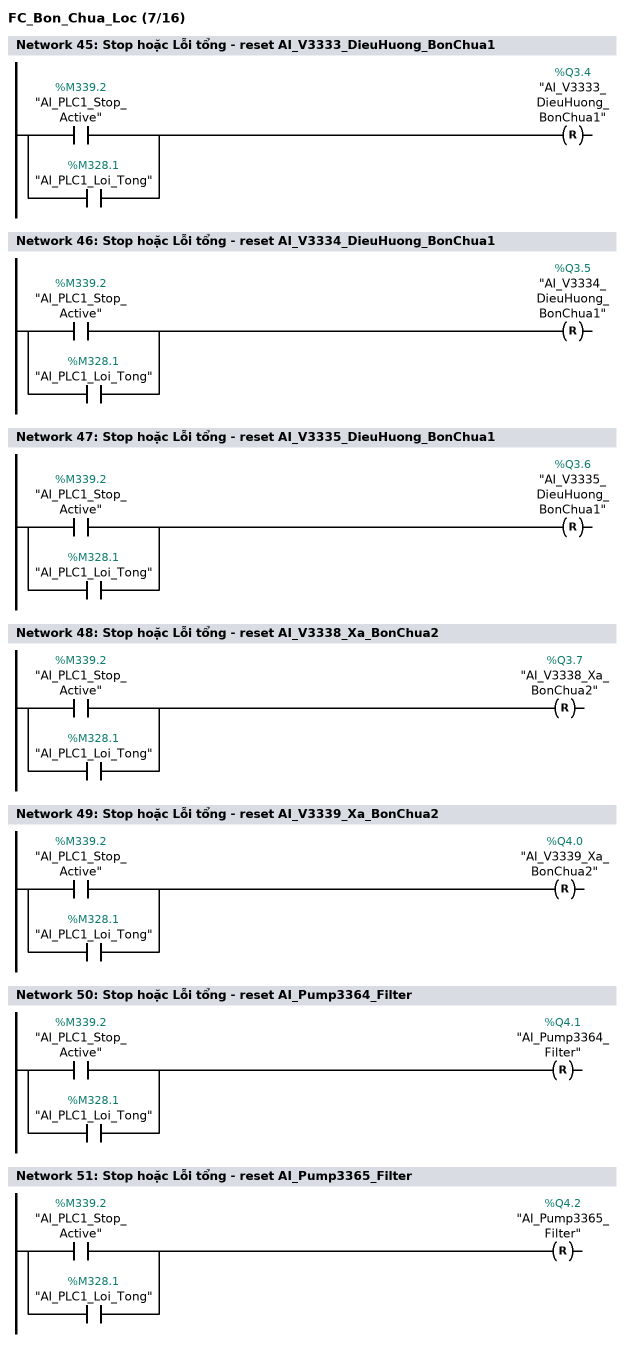
   RUNG wire#powerrail
      Contact( "AI_PLC1_Stop_Active" )
      wire#w1
      R_Coil( "AI_V3333_DieuHuong_BonChua1" )
   END_RUNG
   RUNG wire#powerrail
      Contact( "AI_PLC1_Loi_Tong" )
   END_RUNG wire#w1
   // the same network as SCL:
   IF "AI_PLC1_Stop_Active" OR "AI_PLC1_Loi_Tong" THEN "AI_V3333_DieuHuong_BonChua1" := FALSE; END_IF;
END_REGION

REGION Network 46: Stop hoặc Lỗi tổng - reset AI_V3334_DieuHuong_BonChua1
   RUNG wire#powerrail
      Contact( "AI_PLC1_Stop_Active" )
      wire#w1
      R_Coil( "AI_V3334_DieuHuong_BonChua1" )
   END_RUNG
   RUNG wire#powerrail
      Contact( "AI_PLC1_Loi_Tong" )
   END_RUNG wire#w1
   // the same network as SCL:
   IF "AI_PLC1_Stop_Active" OR "AI_PLC1_Loi_Tong" THEN "AI_V3334_DieuHuong_BonChua1" := FALSE; END_IF;
END_REGION

REGION Network 47: Stop hoặc Lỗi tổng - reset AI_V3335_DieuHuong_BonChua1
   RUNG wire#powerrail
      Contact( "AI_PLC1_Stop_Active" )
      wire#w1
      R_Coil( "AI_V3335_DieuHuong_BonChua1" )
   END_RUNG
   RUNG wire#powerrail
      Contact( "AI_PLC1_Loi_Tong" )
   END_RUNG wire#w1
   // the same network as SCL:
   IF "AI_PLC1_Stop_Active" OR "AI_PLC1_Loi_Tong" THEN "AI_V3335_DieuHuong_BonChua1" := FALSE; END_IF;
END_REGION

REGION Network 48: Stop hoặc Lỗi tổng - reset AI_V3338_Xa_BonChua2
   RUNG wire#powerrail
      Contact( "AI_PLC1_Stop_Active" )
      wire#w1
      R_Coil( "AI_V3338_Xa_BonChua2" )
   END_RUNG
   RUNG wire#powerrail
      Contact( "AI_PLC1_Loi_Tong" )
   END_RUNG wire#w1
   // the same network as SCL:
   IF "AI_PLC1_Stop_Active" OR "AI_PLC1_Loi_Tong" THEN "AI_V3338_Xa_BonChua2" := FALSE; END_IF;
END_REGION

REGION Network 49: Stop hoặc Lỗi tổng - reset AI_V3339_Xa_BonChua2
   RUNG wire#powerrail
      Contact( "AI_PLC1_Stop_Active" )
      wire#w1
      R_Coil( "AI_V3339_Xa_BonChua2" )
   END_RUNG
   RUNG wire#powerrail
      Contact( "AI_PLC1_Loi_Tong" )
   END_RUNG wire#w1
   // the same network as SCL:
   IF "AI_PLC1_Stop_Active" OR "AI_PLC1_Loi_Tong" THEN "AI_V3339_Xa_BonChua2" := FALSE; END_IF;
END_REGION

REGION Network 50: Stop hoặc Lỗi tổng - reset AI_Pump3364_Filter
   RUNG wire#powerrail
      Contact( "AI_PLC1_Stop_Active" )
      wire#w1
      R_Coil( "AI_Pump3364_Filter" )
   END_RUNG
   RUNG wire#powerrail
      Contact( "AI_PLC1_Loi_Tong" )
   END_RUNG wire#w1
   // the same network as SCL:
   IF "AI_PLC1_Stop_Active" OR "AI_PLC1_Loi_Tong" THEN "AI_Pump3364_Filter" := FALSE; END_IF;
END_REGION

REGION Network 51: Stop hoặc Lỗi tổng - reset AI_Pump3365_Filter
   RUNG wire#powerrail
      Contact( "AI_PLC1_Stop_Active" )
      wire#w1
      R_Coil( "AI_Pump3365_Filter" )
   END_RUNG
   RUNG wire#powerrail
      Contact( "AI_PLC1_Loi_Tong" )
   END_RUNG wire#w1
   // the same network as SCL:
   IF "AI_PLC1_Stop_Active" OR "AI_PLC1_Loi_Tong" THEN "AI_Pump3365_Filter" := FALSE; END_IF;
END_REGION

REGION Network 52: Stop hoặc Lỗi tổng - reset AI_V3340_Duong_Filter
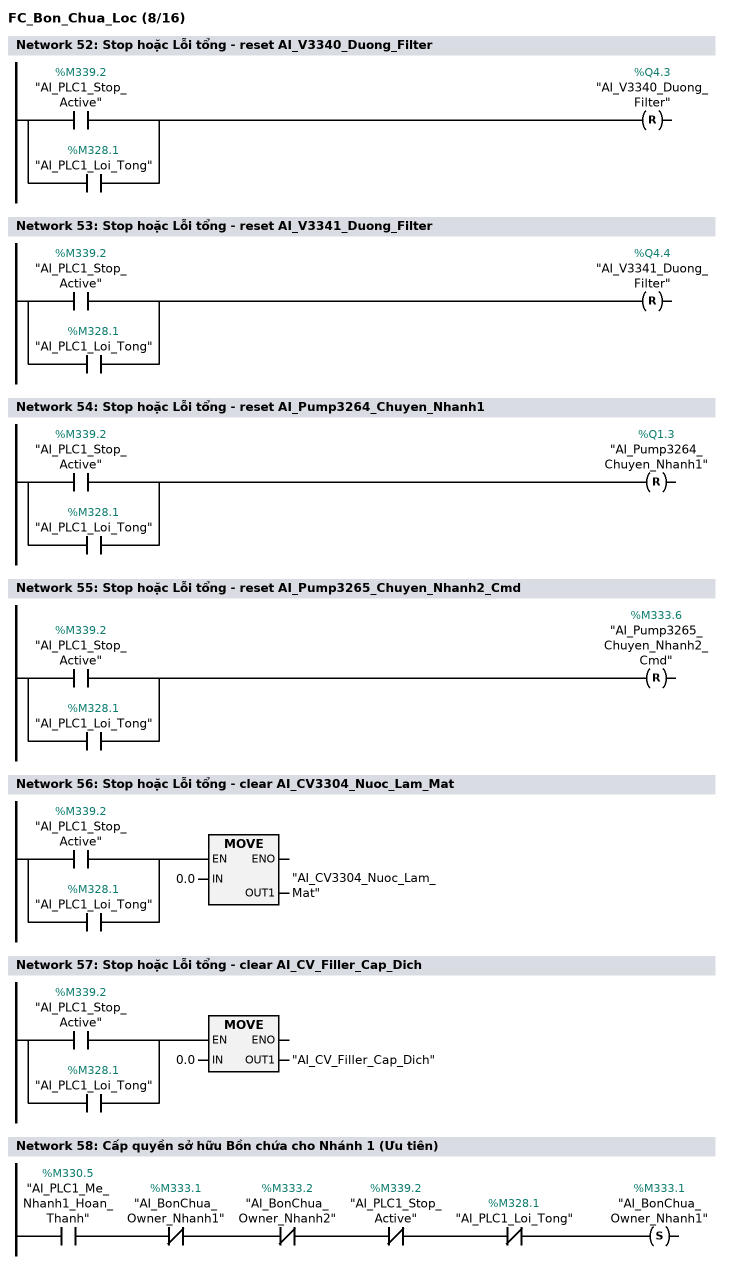
   RUNG wire#powerrail
      Contact( "AI_PLC1_Stop_Active" )
      wire#w1
      R_Coil( "AI_V3340_Duong_Filter" )
   END_RUNG
   RUNG wire#powerrail
      Contact( "AI_PLC1_Loi_Tong" )
   END_RUNG wire#w1
   // the same network as SCL:
   IF "AI_PLC1_Stop_Active" OR "AI_PLC1_Loi_Tong" THEN "AI_V3340_Duong_Filter" := FALSE; END_IF;
END_REGION

REGION Network 53: Stop hoặc Lỗi tổng - reset AI_V3341_Duong_Filter
   RUNG wire#powerrail
      Contact( "AI_PLC1_Stop_Active" )
      wire#w1
      R_Coil( "AI_V3341_Duong_Filter" )
   END_RUNG
   RUNG wire#powerrail
      Contact( "AI_PLC1_Loi_Tong" )
   END_RUNG wire#w1
   // the same network as SCL:
   IF "AI_PLC1_Stop_Active" OR "AI_PLC1_Loi_Tong" THEN "AI_V3341_Duong_Filter" := FALSE; END_IF;
END_REGION

REGION Network 54: Stop hoặc Lỗi tổng - reset AI_Pump3264_Chuyen_Nhanh1
   RUNG wire#powerrail
      Contact( "AI_PLC1_Stop_Active" )
      wire#w1
      R_Coil( "AI_Pump3264_Chuyen_Nhanh1" )
   END_RUNG
   RUNG wire#powerrail
      Contact( "AI_PLC1_Loi_Tong" )
   END_RUNG wire#w1
   // the same network as SCL:
   IF "AI_PLC1_Stop_Active" OR "AI_PLC1_Loi_Tong" THEN "AI_Pump3264_Chuyen_Nhanh1" := FALSE; END_IF;
END_REGION

REGION Network 55: Stop hoặc Lỗi tổng - reset AI_Pump3265_Chuyen_Nhanh2_Cmd
   RUNG wire#powerrail
      Contact( "AI_PLC1_Stop_Active" )
      wire#w1
      R_Coil( "AI_Pump3265_Chuyen_Nhanh2_Cmd" )
   END_RUNG
   RUNG wire#powerrail
      Contact( "AI_PLC1_Loi_Tong" )
   END_RUNG wire#w1
   // the same network as SCL:
   IF "AI_PLC1_Stop_Active" OR "AI_PLC1_Loi_Tong" THEN "AI_Pump3265_Chuyen_Nhanh2_Cmd" := FALSE; END_IF;
END_REGION

REGION Network 56: Stop hoặc Lỗi tổng - clear AI_CV3304_Nuoc_Lam_Mat
   RUNG wire#powerrail
      Contact( "AI_PLC1_Stop_Active" )
      wire#w1
      { S7_GenerateENO := "TRUE" } Move(in := 0.0, out1 => "AI_CV3304_Nuoc_Lam_Mat")
   END_RUNG
   RUNG wire#powerrail
      Contact( "AI_PLC1_Loi_Tong" )
   END_RUNG wire#w1
   // the same network as SCL:
   IF "AI_PLC1_Stop_Active" OR "AI_PLC1_Loi_Tong" THEN "AI_CV3304_Nuoc_Lam_Mat" := 0.0; END_IF;
END_REGION

REGION Network 57: Stop hoặc Lỗi tổng - clear AI_CV_Filler_Cap_Dich
   RUNG wire#powerrail
      Contact( "AI_PLC1_Stop_Active" )
      wire#w1
      { S7_GenerateENO := "TRUE" } Move(in := 0.0, out1 => "AI_CV_Filler_Cap_Dich")
   END_RUNG
   RUNG wire#powerrail
      Contact( "AI_PLC1_Loi_Tong" )
   END_RUNG wire#w1
   // the same network as SCL:
   IF "AI_PLC1_Stop_Active" OR "AI_PLC1_Loi_Tong" THEN "AI_CV_Filler_Cap_Dich" := 0.0; END_IF;
END_REGION

REGION Network 58: Cấp quyền sở hữu Bồn chứa cho Nhánh 1 (Ưu tiên)
   RUNG wire#powerrail
      Contact( "AI_PLC1_Me_Nhanh1_Hoan_Thanh" )
      I_Contact( "AI_BonChua_Owner_Nhanh1" )
      I_Contact( "AI_BonChua_Owner_Nhanh2" )
      I_Contact( "AI_PLC1_Stop_Active" )
      I_Contact( "AI_PLC1_Loi_Tong" )
      S_Coil( "AI_BonChua_Owner_Nhanh1" )
   END_RUNG
   // the same network as SCL:
   IF "AI_PLC1_Me_Nhanh1_Hoan_Thanh" AND NOT "AI_BonChua_Owner_Nhanh1" AND NOT "AI_BonChua_Owner_Nhanh2" AND NOT "AI_PLC1_Stop_Active" AND NOT "AI_PLC1_Loi_Tong" THEN
       "AI_BonChua_Owner_Nhanh1" := TRUE;
   END_IF;
END_REGION

REGION Network 59: Cấp quyền sở hữu Bồn chứa cho Nhánh 2
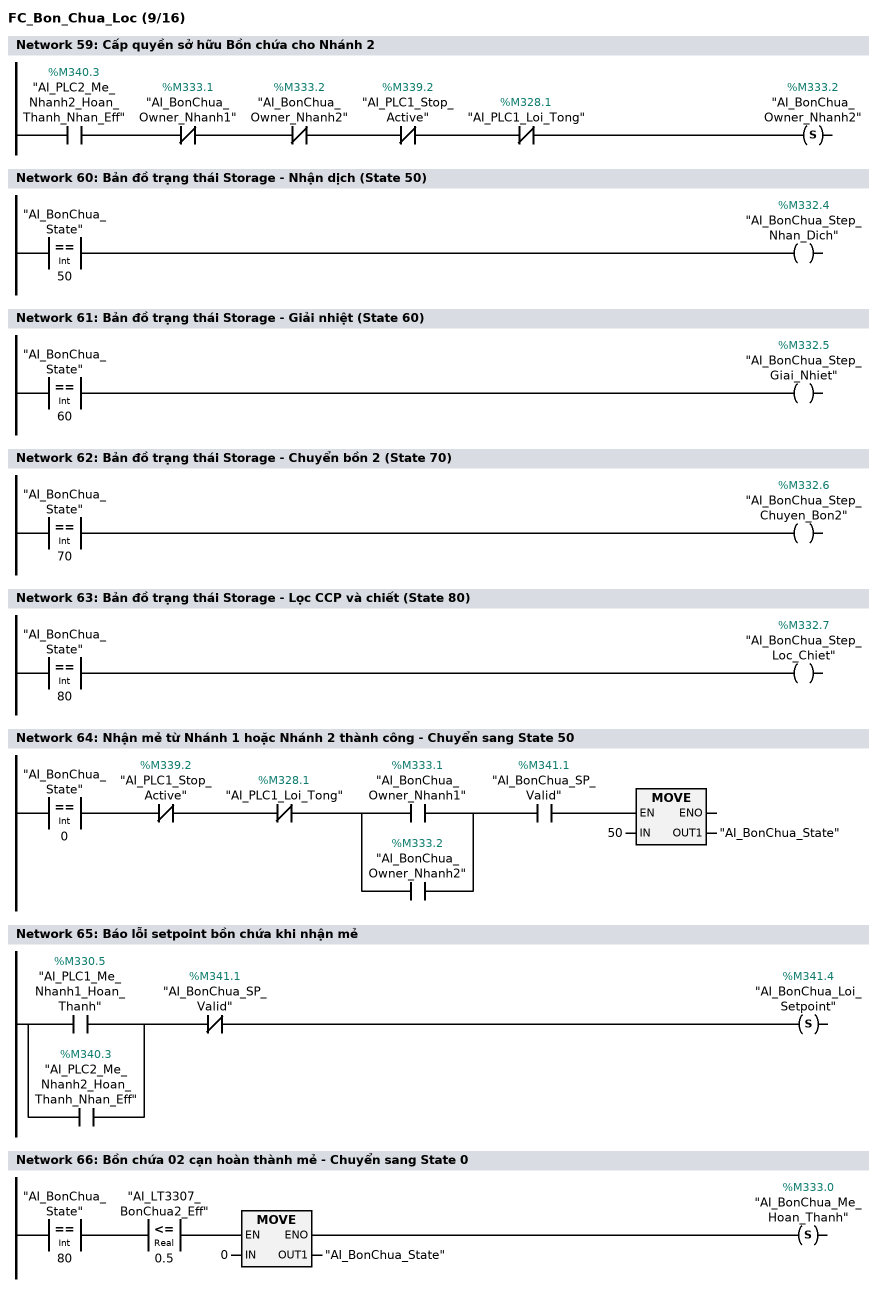
   RUNG wire#powerrail
      Contact( "AI_PLC2_Me_Nhanh2_Hoan_Thanh_Nhan_Eff" )
      I_Contact( "AI_BonChua_Owner_Nhanh1" )
      I_Contact( "AI_BonChua_Owner_Nhanh2" )
      I_Contact( "AI_PLC1_Stop_Active" )
      I_Contact( "AI_PLC1_Loi_Tong" )
      S_Coil( "AI_BonChua_Owner_Nhanh2" )
   END_RUNG
   // the same network as SCL:
   IF "AI_PLC2_Me_Nhanh2_Hoan_Thanh_Nhan_Eff" AND NOT "AI_BonChua_Owner_Nhanh1" AND NOT "AI_BonChua_Owner_Nhanh2" AND NOT "AI_PLC1_Stop_Active" AND NOT "AI_PLC1_Loi_Tong" THEN
       "AI_BonChua_Owner_Nhanh2" := TRUE;
   END_IF;
END_REGION

REGION Network 60: Bản đồ trạng thái Storage - Nhận dịch (State 50)
   RUNG wire#powerrail
      { S7_Templates := "SrcType := Int" } EQ_Contact(in1 := "AI_BonChua_State", in2 := 50)
      Coil( "AI_BonChua_Step_Nhan_Dich" )
   END_RUNG
   // the same network as SCL:
   "AI_BonChua_Step_Nhan_Dich" := "AI_BonChua_State" = 50;
END_REGION

REGION Network 61: Bản đồ trạng thái Storage - Giải nhiệt (State 60)
   RUNG wire#powerrail
      { S7_Templates := "SrcType := Int" } EQ_Contact(in1 := "AI_BonChua_State", in2 := 60)
      Coil( "AI_BonChua_Step_Giai_Nhiet" )
   END_RUNG
   // the same network as SCL:
   "AI_BonChua_Step_Giai_Nhiet" := "AI_BonChua_State" = 60;
END_REGION

REGION Network 62: Bản đồ trạng thái Storage - Chuyển bồn 2 (State 70)
   RUNG wire#powerrail
      { S7_Templates := "SrcType := Int" } EQ_Contact(in1 := "AI_BonChua_State", in2 := 70)
      Coil( "AI_BonChua_Step_Chuyen_Bon2" )
   END_RUNG
   // the same network as SCL:
   "AI_BonChua_Step_Chuyen_Bon2" := "AI_BonChua_State" = 70;
END_REGION

REGION Network 63: Bản đồ trạng thái Storage - Lọc CCP và chiết (State 80)
   RUNG wire#powerrail
      { S7_Templates := "SrcType := Int" } EQ_Contact(in1 := "AI_BonChua_State", in2 := 80)
      Coil( "AI_BonChua_Step_Loc_Chiet" )
   END_RUNG
   // the same network as SCL:
   "AI_BonChua_Step_Loc_Chiet" := "AI_BonChua_State" = 80;
END_REGION

REGION Network 64: Nhận mẻ từ Nhánh 1 hoặc Nhánh 2 thành công - Chuyển sang State 50
   RUNG wire#powerrail
      { S7_Templates := "SrcType := Int" } EQ_Contact(in1 := "AI_BonChua_State", in2 := 0)
      I_Contact( "AI_PLC1_Stop_Active" )
      I_Contact( "AI_PLC1_Loi_Tong" )
      wire#w1
      Contact( "AI_BonChua_Owner_Nhanh1" )
      wire#w2
      Contact( "AI_BonChua_SP_Valid" )
      { S7_GenerateENO := "TRUE" } Move(in := 50, out1 => "AI_BonChua_State")
   END_RUNG
   RUNG wire#w1
      Contact( "AI_BonChua_Owner_Nhanh2" )
   END_RUNG wire#w2
   // the same network as SCL:
   IF ("AI_BonChua_State" = 0) AND NOT "AI_PLC1_Stop_Active" AND NOT "AI_PLC1_Loi_Tong" AND ("AI_BonChua_Owner_Nhanh1" OR "AI_BonChua_Owner_Nhanh2") AND "AI_BonChua_SP_Valid" THEN
       "AI_BonChua_State" := 50;
   END_IF;
END_REGION

REGION Network 65: Báo lỗi setpoint bồn chứa khi nhận mẻ
   RUNG wire#powerrail
      Contact( "AI_PLC1_Me_Nhanh1_Hoan_Thanh" )
      wire#w1
      I_Contact( "AI_BonChua_SP_Valid" )
      S_Coil( "AI_BonChua_Loi_Setpoint" )
   END_RUNG
   RUNG wire#powerrail
      Contact( "AI_PLC2_Me_Nhanh2_Hoan_Thanh_Nhan_Eff" )
   END_RUNG wire#w1
   // the same network as SCL:
   IF ("AI_PLC1_Me_Nhanh1_Hoan_Thanh" OR "AI_PLC2_Me_Nhanh2_Hoan_Thanh_Nhan_Eff") AND NOT "AI_BonChua_SP_Valid" THEN
       "AI_BonChua_Loi_Setpoint" := TRUE;
   END_IF;
END_REGION

REGION Network 66: Bồn chứa 02 cạn hoàn thành mẻ - Chuyển sang State 0
   RUNG wire#powerrail
      { S7_Templates := "SrcType := Int" } EQ_Contact(in1 := "AI_BonChua_State", in2 := 80)
      { S7_Templates := "SrcType := Real" } LE_Contact(in1 := "AI_LT3307_BonChua2_Eff", in2 := 0.5)
      { S7_GenerateENO := "TRUE" } Move(in := 0, out1 => "AI_BonChua_State")
      S_Coil( "AI_BonChua_Me_Hoan_Thanh" )
   END_RUNG
   // the same network as SCL:
   // ENO of a box is taken as its EN; it also drops when the box reports an error
   #_w1 := ("AI_BonChua_State" = 80) AND ("AI_LT3307_BonChua2_Eff" <= 0.5);
   IF #_w1 THEN
       "AI_BonChua_State" := 0;
       "AI_BonChua_Me_Hoan_Thanh" := TRUE;
   END_IF;
END_REGION

REGION Network 67: Chuyển sang Bồn chứa 02 xong - Chuyển sang State 80
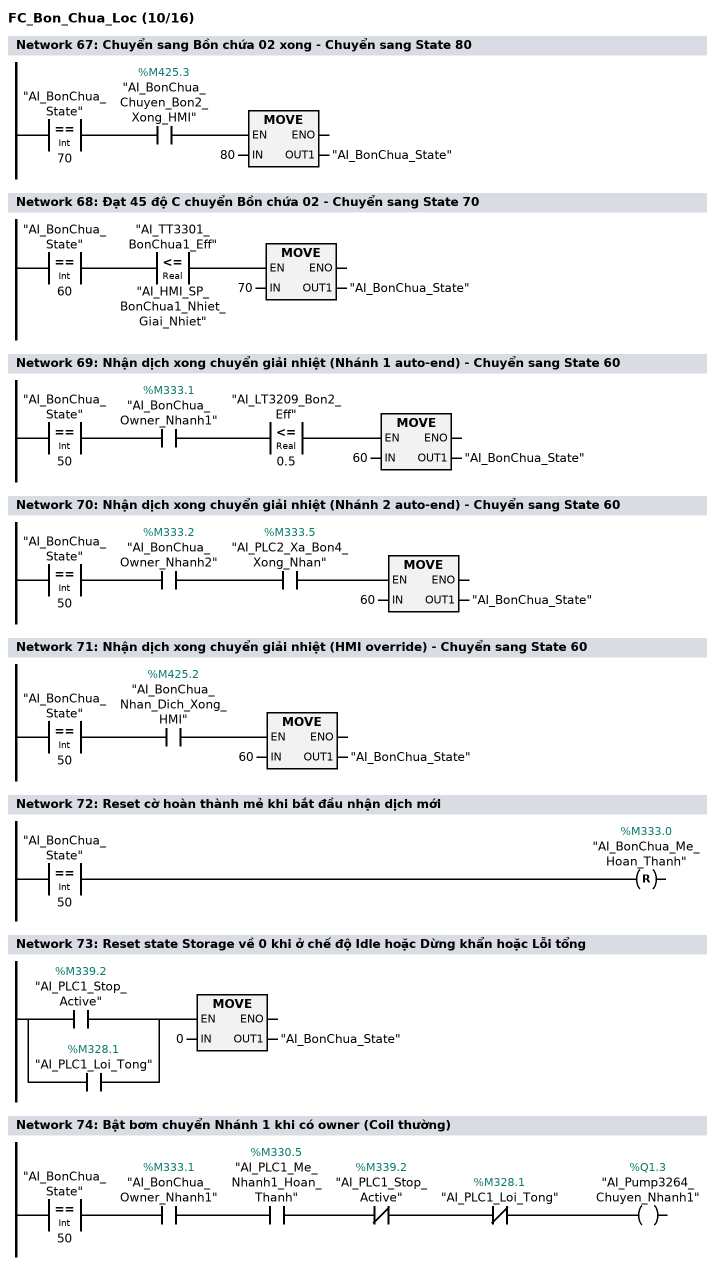
   RUNG wire#powerrail
      { S7_Templates := "SrcType := Int" } EQ_Contact(in1 := "AI_BonChua_State", in2 := 70)
      Contact( "AI_BonChua_Chuyen_Bon2_Xong_HMI" )
      { S7_GenerateENO := "TRUE" } Move(in := 80, out1 => "AI_BonChua_State")
   END_RUNG
   // the same network as SCL:
   IF ("AI_BonChua_State" = 70) AND "AI_BonChua_Chuyen_Bon2_Xong_HMI" THEN "AI_BonChua_State" := 80; END_IF;
END_REGION

REGION Network 68: Đạt 45 độ C chuyển Bồn chứa 02 - Chuyển sang State 70
   RUNG wire#powerrail
      { S7_Templates := "SrcType := Int" } EQ_Contact(in1 := "AI_BonChua_State", in2 := 60)
      { S7_Templates := "SrcType := Real" } LE_Contact(in1 := "AI_TT3301_BonChua1_Eff", in2 := "AI_HMI_SP_BonChua1_Nhiet_Giai_Nhiet")
      { S7_GenerateENO := "TRUE" } Move(in := 70, out1 => "AI_BonChua_State")
   END_RUNG
   // the same network as SCL:
   IF ("AI_BonChua_State" = 60) AND ("AI_TT3301_BonChua1_Eff" <= "AI_HMI_SP_BonChua1_Nhiet_Giai_Nhiet") THEN
       "AI_BonChua_State" := 70;
   END_IF;
END_REGION

REGION Network 69: Nhận dịch xong chuyển giải nhiệt (Nhánh 1 auto-end) - Chuyển sang State 60
   RUNG wire#powerrail
      { S7_Templates := "SrcType := Int" } EQ_Contact(in1 := "AI_BonChua_State", in2 := 50)
      Contact( "AI_BonChua_Owner_Nhanh1" )
      { S7_Templates := "SrcType := Real" } LE_Contact(in1 := "AI_LT3209_Bon2_Eff", in2 := 0.5)
      { S7_GenerateENO := "TRUE" } Move(in := 60, out1 => "AI_BonChua_State")
   END_RUNG
   // the same network as SCL:
   IF ("AI_BonChua_State" = 50) AND "AI_BonChua_Owner_Nhanh1" AND ("AI_LT3209_Bon2_Eff" <= 0.5) THEN
       "AI_BonChua_State" := 60;
   END_IF;
END_REGION

REGION Network 70: Nhận dịch xong chuyển giải nhiệt (Nhánh 2 auto-end) - Chuyển sang State 60
   RUNG wire#powerrail
      { S7_Templates := "SrcType := Int" } EQ_Contact(in1 := "AI_BonChua_State", in2 := 50)
      Contact( "AI_BonChua_Owner_Nhanh2" )
      Contact( "AI_PLC2_Xa_Bon4_Xong_Nhan" )
      { S7_GenerateENO := "TRUE" } Move(in := 60, out1 => "AI_BonChua_State")
   END_RUNG
   // the same network as SCL:
   IF ("AI_BonChua_State" = 50) AND "AI_BonChua_Owner_Nhanh2" AND "AI_PLC2_Xa_Bon4_Xong_Nhan" THEN
       "AI_BonChua_State" := 60;
   END_IF;
END_REGION

REGION Network 71: Nhận dịch xong chuyển giải nhiệt (HMI override) - Chuyển sang State 60
   RUNG wire#powerrail
      { S7_Templates := "SrcType := Int" } EQ_Contact(in1 := "AI_BonChua_State", in2 := 50)
      Contact( "AI_BonChua_Nhan_Dich_Xong_HMI" )
      { S7_GenerateENO := "TRUE" } Move(in := 60, out1 => "AI_BonChua_State")
   END_RUNG
   // the same network as SCL:
   IF ("AI_BonChua_State" = 50) AND "AI_BonChua_Nhan_Dich_Xong_HMI" THEN "AI_BonChua_State" := 60; END_IF;
END_REGION

REGION Network 72: Reset cờ hoàn thành mẻ khi bắt đầu nhận dịch mới
   RUNG wire#powerrail
      { S7_Templates := "SrcType := Int" } EQ_Contact(in1 := "AI_BonChua_State", in2 := 50)
      R_Coil( "AI_BonChua_Me_Hoan_Thanh" )
   END_RUNG
   // the same network as SCL:
   IF "AI_BonChua_State" = 50 THEN "AI_BonChua_Me_Hoan_Thanh" := FALSE; END_IF;
END_REGION

REGION Network 73: Reset state Storage về 0 khi ở chế độ Idle hoặc Dừng khẩn hoặc Lỗi tổng
   RUNG wire#powerrail
      Contact( "AI_PLC1_Stop_Active" )
      wire#w1
      { S7_GenerateENO := "TRUE" } Move(in := 0, out1 => "AI_BonChua_State")
   END_RUNG
   RUNG wire#powerrail
      Contact( "AI_PLC1_Loi_Tong" )
   END_RUNG wire#w1
   // the same network as SCL:
   IF "AI_PLC1_Stop_Active" OR "AI_PLC1_Loi_Tong" THEN "AI_BonChua_State" := 0; END_IF;
END_REGION

REGION Network 74: Bật bơm chuyển Nhánh 1 khi có owner (Coil thường)
   RUNG wire#powerrail
      { S7_Templates := "SrcType := Int" } EQ_Contact(in1 := "AI_BonChua_State", in2 := 50)
      Contact( "AI_BonChua_Owner_Nhanh1" )
      Contact( "AI_PLC1_Me_Nhanh1_Hoan_Thanh" )
      I_Contact( "AI_PLC1_Stop_Active" )
      I_Contact( "AI_PLC1_Loi_Tong" )
      Coil( "AI_Pump3264_Chuyen_Nhanh1" )
   END_RUNG
   // the same network as SCL:
   "AI_Pump3264_Chuyen_Nhanh1" := ("AI_BonChua_State" = 50) AND "AI_BonChua_Owner_Nhanh1" AND "AI_PLC1_Me_Nhanh1_Hoan_Thanh" AND NOT "AI_PLC1_Stop_Active" AND NOT "AI_PLC1_Loi_Tong";
END_REGION

REGION Network 75: Bật bơm chuyển Nhánh 2 khi có owner (Coil thường)
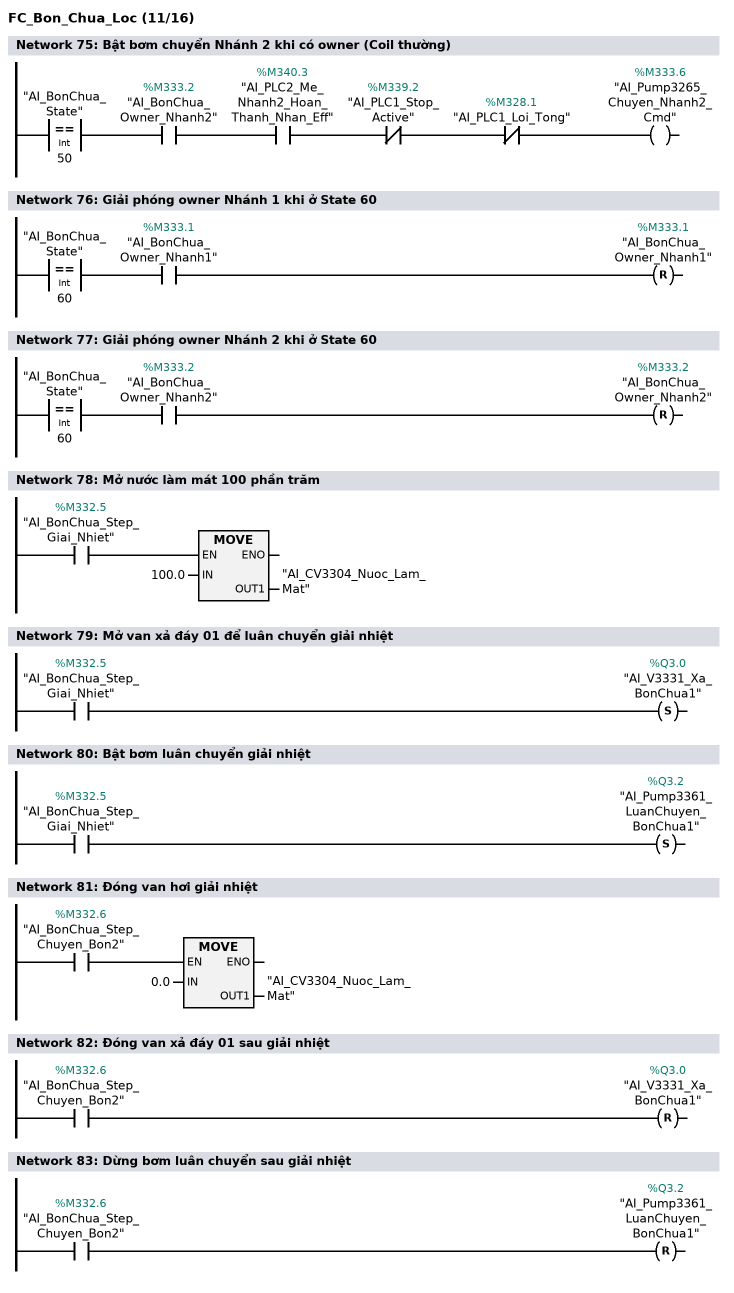
   RUNG wire#powerrail
      { S7_Templates := "SrcType := Int" } EQ_Contact(in1 := "AI_BonChua_State", in2 := 50)
      Contact( "AI_BonChua_Owner_Nhanh2" )
      Contact( "AI_PLC2_Me_Nhanh2_Hoan_Thanh_Nhan_Eff" )
      I_Contact( "AI_PLC1_Stop_Active" )
      I_Contact( "AI_PLC1_Loi_Tong" )
      Coil( "AI_Pump3265_Chuyen_Nhanh2_Cmd" )
   END_RUNG
   // the same network as SCL:
   "AI_Pump3265_Chuyen_Nhanh2_Cmd" := ("AI_BonChua_State" = 50) AND "AI_BonChua_Owner_Nhanh2" AND "AI_PLC2_Me_Nhanh2_Hoan_Thanh_Nhan_Eff" AND NOT "AI_PLC1_Stop_Active" AND NOT "AI_PLC1_Loi_Tong";
END_REGION

REGION Network 76: Giải phóng owner Nhánh 1 khi ở State 60
   RUNG wire#powerrail
      { S7_Templates := "SrcType := Int" } EQ_Contact(in1 := "AI_BonChua_State", in2 := 60)
      Contact( "AI_BonChua_Owner_Nhanh1" )
      R_Coil( "AI_BonChua_Owner_Nhanh1" )
   END_RUNG
   // the same network as SCL:
   IF ("AI_BonChua_State" = 60) AND "AI_BonChua_Owner_Nhanh1" THEN
       "AI_BonChua_Owner_Nhanh1" := FALSE;
   END_IF;
END_REGION

REGION Network 77: Giải phóng owner Nhánh 2 khi ở State 60
   RUNG wire#powerrail
      { S7_Templates := "SrcType := Int" } EQ_Contact(in1 := "AI_BonChua_State", in2 := 60)
      Contact( "AI_BonChua_Owner_Nhanh2" )
      R_Coil( "AI_BonChua_Owner_Nhanh2" )
   END_RUNG
   // the same network as SCL:
   IF ("AI_BonChua_State" = 60) AND "AI_BonChua_Owner_Nhanh2" THEN
       "AI_BonChua_Owner_Nhanh2" := FALSE;
   END_IF;
END_REGION

REGION Network 78: Mở nước làm mát 100 phần trăm
   RUNG wire#powerrail
      Contact( "AI_BonChua_Step_Giai_Nhiet" )
      { S7_GenerateENO := "TRUE" } Move(in := 100.0, out1 => "AI_CV3304_Nuoc_Lam_Mat")
   END_RUNG
   // the same network as SCL:
   IF "AI_BonChua_Step_Giai_Nhiet" THEN "AI_CV3304_Nuoc_Lam_Mat" := 100.0; END_IF;
END_REGION

REGION Network 79: Mở van xả đáy 01 để luân chuyển giải nhiệt
   RUNG wire#powerrail
      Contact( "AI_BonChua_Step_Giai_Nhiet" )
      S_Coil( "AI_V3331_Xa_BonChua1" )
   END_RUNG
   // the same network as SCL:
   IF "AI_BonChua_Step_Giai_Nhiet" THEN "AI_V3331_Xa_BonChua1" := TRUE; END_IF;
END_REGION

REGION Network 80: Bật bơm luân chuyển giải nhiệt
   RUNG wire#powerrail
      Contact( "AI_BonChua_Step_Giai_Nhiet" )
      S_Coil( "AI_Pump3361_LuanChuyen_BonChua1" )
   END_RUNG
   // the same network as SCL:
   IF "AI_BonChua_Step_Giai_Nhiet" THEN "AI_Pump3361_LuanChuyen_BonChua1" := TRUE; END_IF;
END_REGION

REGION Network 81: Đóng van hơi giải nhiệt
   RUNG wire#powerrail
      Contact( "AI_BonChua_Step_Chuyen_Bon2" )
      { S7_GenerateENO := "TRUE" } Move(in := 0.0, out1 => "AI_CV3304_Nuoc_Lam_Mat")
   END_RUNG
   // the same network as SCL:
   IF "AI_BonChua_Step_Chuyen_Bon2" THEN "AI_CV3304_Nuoc_Lam_Mat" := 0.0; END_IF;
END_REGION

REGION Network 82: Đóng van xả đáy 01 sau giải nhiệt
   RUNG wire#powerrail
      Contact( "AI_BonChua_Step_Chuyen_Bon2" )
      R_Coil( "AI_V3331_Xa_BonChua1" )
   END_RUNG
   // the same network as SCL:
   IF "AI_BonChua_Step_Chuyen_Bon2" THEN "AI_V3331_Xa_BonChua1" := FALSE; END_IF;
END_REGION

REGION Network 83: Dừng bơm luân chuyển sau giải nhiệt
   RUNG wire#powerrail
      Contact( "AI_BonChua_Step_Chuyen_Bon2" )
      R_Coil( "AI_Pump3361_LuanChuyen_BonChua1" )
   END_RUNG
   // the same network as SCL:
   IF "AI_BonChua_Step_Chuyen_Bon2" THEN "AI_Pump3361_LuanChuyen_BonChua1" := FALSE; END_IF;
END_REGION

REGION Network 84: Mở van xả đáy 02 để chuyển bồn
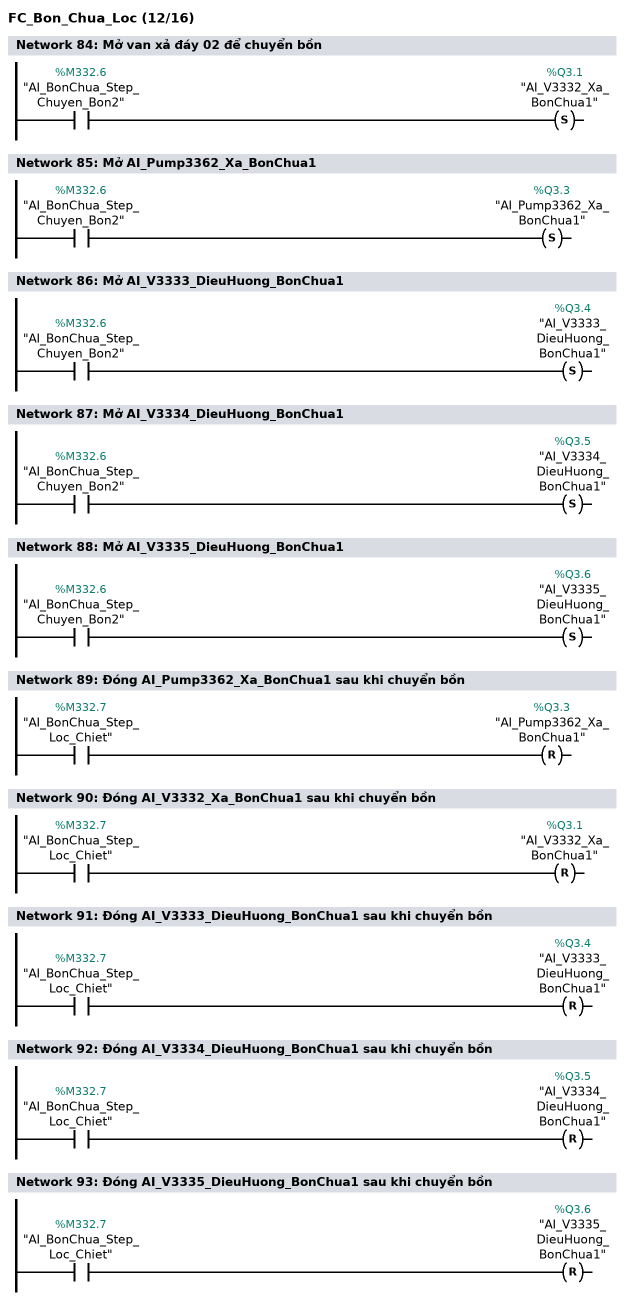
   RUNG wire#powerrail
      Contact( "AI_BonChua_Step_Chuyen_Bon2" )
      S_Coil( "AI_V3332_Xa_BonChua1" )
   END_RUNG
   // the same network as SCL:
   IF "AI_BonChua_Step_Chuyen_Bon2" THEN "AI_V3332_Xa_BonChua1" := TRUE; END_IF;
END_REGION

REGION Network 85: Mở AI_Pump3362_Xa_BonChua1
   RUNG wire#powerrail
      Contact( "AI_BonChua_Step_Chuyen_Bon2" )
      S_Coil( "AI_Pump3362_Xa_BonChua1" )
   END_RUNG
   // the same network as SCL:
   IF "AI_BonChua_Step_Chuyen_Bon2" THEN "AI_Pump3362_Xa_BonChua1" := TRUE; END_IF;
END_REGION

REGION Network 86: Mở AI_V3333_DieuHuong_BonChua1
   RUNG wire#powerrail
      Contact( "AI_BonChua_Step_Chuyen_Bon2" )
      S_Coil( "AI_V3333_DieuHuong_BonChua1" )
   END_RUNG
   // the same network as SCL:
   IF "AI_BonChua_Step_Chuyen_Bon2" THEN "AI_V3333_DieuHuong_BonChua1" := TRUE; END_IF;
END_REGION

REGION Network 87: Mở AI_V3334_DieuHuong_BonChua1
   RUNG wire#powerrail
      Contact( "AI_BonChua_Step_Chuyen_Bon2" )
      S_Coil( "AI_V3334_DieuHuong_BonChua1" )
   END_RUNG
   // the same network as SCL:
   IF "AI_BonChua_Step_Chuyen_Bon2" THEN "AI_V3334_DieuHuong_BonChua1" := TRUE; END_IF;
END_REGION

REGION Network 88: Mở AI_V3335_DieuHuong_BonChua1
   RUNG wire#powerrail
      Contact( "AI_BonChua_Step_Chuyen_Bon2" )
      S_Coil( "AI_V3335_DieuHuong_BonChua1" )
   END_RUNG
   // the same network as SCL:
   IF "AI_BonChua_Step_Chuyen_Bon2" THEN "AI_V3335_DieuHuong_BonChua1" := TRUE; END_IF;
END_REGION

REGION Network 89: Đóng AI_Pump3362_Xa_BonChua1 sau khi chuyển bồn
   RUNG wire#powerrail
      Contact( "AI_BonChua_Step_Loc_Chiet" )
      R_Coil( "AI_Pump3362_Xa_BonChua1" )
   END_RUNG
   // the same network as SCL:
   IF "AI_BonChua_Step_Loc_Chiet" THEN "AI_Pump3362_Xa_BonChua1" := FALSE; END_IF;
END_REGION

REGION Network 90: Đóng AI_V3332_Xa_BonChua1 sau khi chuyển bồn
   RUNG wire#powerrail
      Contact( "AI_BonChua_Step_Loc_Chiet" )
      R_Coil( "AI_V3332_Xa_BonChua1" )
   END_RUNG
   // the same network as SCL:
   IF "AI_BonChua_Step_Loc_Chiet" THEN "AI_V3332_Xa_BonChua1" := FALSE; END_IF;
END_REGION

REGION Network 91: Đóng AI_V3333_DieuHuong_BonChua1 sau khi chuyển bồn
   RUNG wire#powerrail
      Contact( "AI_BonChua_Step_Loc_Chiet" )
      R_Coil( "AI_V3333_DieuHuong_BonChua1" )
   END_RUNG
   // the same network as SCL:
   IF "AI_BonChua_Step_Loc_Chiet" THEN "AI_V3333_DieuHuong_BonChua1" := FALSE; END_IF;
END_REGION

REGION Network 92: Đóng AI_V3334_DieuHuong_BonChua1 sau khi chuyển bồn
   RUNG wire#powerrail
      Contact( "AI_BonChua_Step_Loc_Chiet" )
      R_Coil( "AI_V3334_DieuHuong_BonChua1" )
   END_RUNG
   // the same network as SCL:
   IF "AI_BonChua_Step_Loc_Chiet" THEN "AI_V3334_DieuHuong_BonChua1" := FALSE; END_IF;
END_REGION

REGION Network 93: Đóng AI_V3335_DieuHuong_BonChua1 sau khi chuyển bồn
   RUNG wire#powerrail
      Contact( "AI_BonChua_Step_Loc_Chiet" )
      R_Coil( "AI_V3335_DieuHuong_BonChua1" )
   END_RUNG
   // the same network as SCL:
   IF "AI_BonChua_Step_Loc_Chiet" THEN "AI_V3335_DieuHuong_BonChua1" := FALSE; END_IF;
END_REGION

REGION Network 94: Chạy AI_Pump3364_Filter (Coil thường)
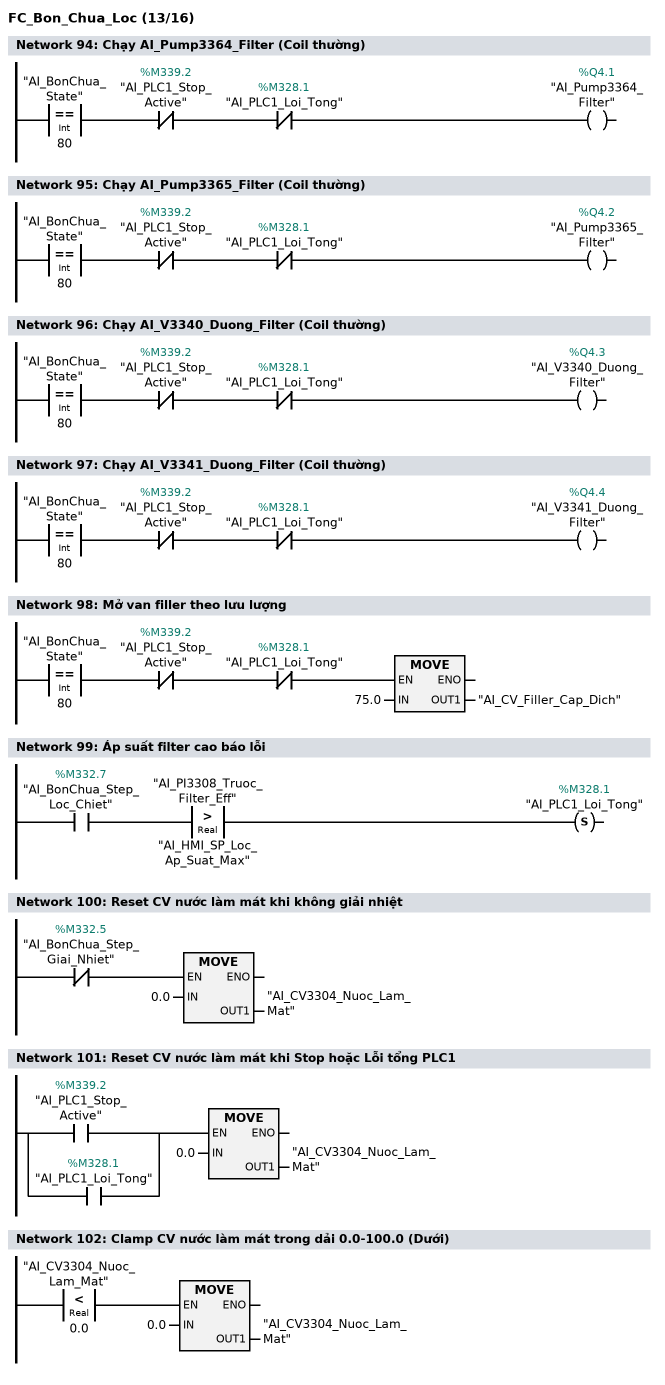
   RUNG wire#powerrail
      { S7_Templates := "SrcType := Int" } EQ_Contact(in1 := "AI_BonChua_State", in2 := 80)
      I_Contact( "AI_PLC1_Stop_Active" )
      I_Contact( "AI_PLC1_Loi_Tong" )
      Coil( "AI_Pump3364_Filter" )
   END_RUNG
   // the same network as SCL:
   "AI_Pump3364_Filter" := ("AI_BonChua_State" = 80) AND NOT "AI_PLC1_Stop_Active" AND NOT "AI_PLC1_Loi_Tong";
END_REGION

REGION Network 95: Chạy AI_Pump3365_Filter (Coil thường)
   RUNG wire#powerrail
      { S7_Templates := "SrcType := Int" } EQ_Contact(in1 := "AI_BonChua_State", in2 := 80)
      I_Contact( "AI_PLC1_Stop_Active" )
      I_Contact( "AI_PLC1_Loi_Tong" )
      Coil( "AI_Pump3365_Filter" )
   END_RUNG
   // the same network as SCL:
   "AI_Pump3365_Filter" := ("AI_BonChua_State" = 80) AND NOT "AI_PLC1_Stop_Active" AND NOT "AI_PLC1_Loi_Tong";
END_REGION

REGION Network 96: Chạy AI_V3340_Duong_Filter (Coil thường)
   RUNG wire#powerrail
      { S7_Templates := "SrcType := Int" } EQ_Contact(in1 := "AI_BonChua_State", in2 := 80)
      I_Contact( "AI_PLC1_Stop_Active" )
      I_Contact( "AI_PLC1_Loi_Tong" )
      Coil( "AI_V3340_Duong_Filter" )
   END_RUNG
   // the same network as SCL:
   "AI_V3340_Duong_Filter" := ("AI_BonChua_State" = 80) AND NOT "AI_PLC1_Stop_Active" AND NOT "AI_PLC1_Loi_Tong";
END_REGION

REGION Network 97: Chạy AI_V3341_Duong_Filter (Coil thường)
   RUNG wire#powerrail
      { S7_Templates := "SrcType := Int" } EQ_Contact(in1 := "AI_BonChua_State", in2 := 80)
      I_Contact( "AI_PLC1_Stop_Active" )
      I_Contact( "AI_PLC1_Loi_Tong" )
      Coil( "AI_V3341_Duong_Filter" )
   END_RUNG
   // the same network as SCL:
   "AI_V3341_Duong_Filter" := ("AI_BonChua_State" = 80) AND NOT "AI_PLC1_Stop_Active" AND NOT "AI_PLC1_Loi_Tong";
END_REGION

REGION Network 98: Mở van filler theo lưu lượng
   RUNG wire#powerrail
      { S7_Templates := "SrcType := Int" } EQ_Contact(in1 := "AI_BonChua_State", in2 := 80)
      I_Contact( "AI_PLC1_Stop_Active" )
      I_Contact( "AI_PLC1_Loi_Tong" )
      { S7_GenerateENO := "TRUE" } Move(in := 75.0, out1 => "AI_CV_Filler_Cap_Dich")
   END_RUNG
   // the same network as SCL:
   IF ("AI_BonChua_State" = 80) AND NOT "AI_PLC1_Stop_Active" AND NOT "AI_PLC1_Loi_Tong" THEN
       "AI_CV_Filler_Cap_Dich" := 75.0;
   END_IF;
END_REGION

REGION Network 99: Áp suất filter cao báo lỗi
   RUNG wire#powerrail
      Contact( "AI_BonChua_Step_Loc_Chiet" )
      { S7_Templates := "SrcType := Real" } GT_Contact(in1 := "AI_PI3308_Truoc_Filter_Eff", in2 := "AI_HMI_SP_Loc_Ap_Suat_Max")
      S_Coil( "AI_PLC1_Loi_Tong" )
   END_RUNG
   // the same network as SCL:
   IF "AI_BonChua_Step_Loc_Chiet" AND ("AI_PI3308_Truoc_Filter_Eff" > "AI_HMI_SP_Loc_Ap_Suat_Max") THEN
       "AI_PLC1_Loi_Tong" := TRUE;
   END_IF;
END_REGION

REGION Network 100: Reset CV nước làm mát khi không giải nhiệt
   RUNG wire#powerrail
      I_Contact( "AI_BonChua_Step_Giai_Nhiet" )
      { S7_GenerateENO := "TRUE" } Move(in := 0.0, out1 => "AI_CV3304_Nuoc_Lam_Mat")
   END_RUNG
   // the same network as SCL:
   IF NOT "AI_BonChua_Step_Giai_Nhiet" THEN "AI_CV3304_Nuoc_Lam_Mat" := 0.0; END_IF;
END_REGION

REGION Network 101: Reset CV nước làm mát khi Stop hoặc Lỗi tổng PLC1
   RUNG wire#powerrail
      Contact( "AI_PLC1_Stop_Active" )
      wire#w1
      { S7_GenerateENO := "TRUE" } Move(in := 0.0, out1 => "AI_CV3304_Nuoc_Lam_Mat")
   END_RUNG
   RUNG wire#powerrail
      Contact( "AI_PLC1_Loi_Tong" )
   END_RUNG wire#w1
   // the same network as SCL:
   IF "AI_PLC1_Stop_Active" OR "AI_PLC1_Loi_Tong" THEN "AI_CV3304_Nuoc_Lam_Mat" := 0.0; END_IF;
END_REGION

REGION Network 102: Clamp CV nước làm mát trong dải 0.0-100.0 (Dưới)
   RUNG wire#powerrail
      { S7_Templates := "SrcType := Real" } LT_Contact(in1 := "AI_CV3304_Nuoc_Lam_Mat", in2 := 0.0)
      { S7_GenerateENO := "TRUE" } Move(in := 0.0, out1 => "AI_CV3304_Nuoc_Lam_Mat")
   END_RUNG
   // the same network as SCL:
   IF "AI_CV3304_Nuoc_Lam_Mat" < 0.0 THEN "AI_CV3304_Nuoc_Lam_Mat" := 0.0; END_IF;
END_REGION

REGION Network 103: Clamp CV nước làm mát trong dải 0.0-100.0 (Trên)
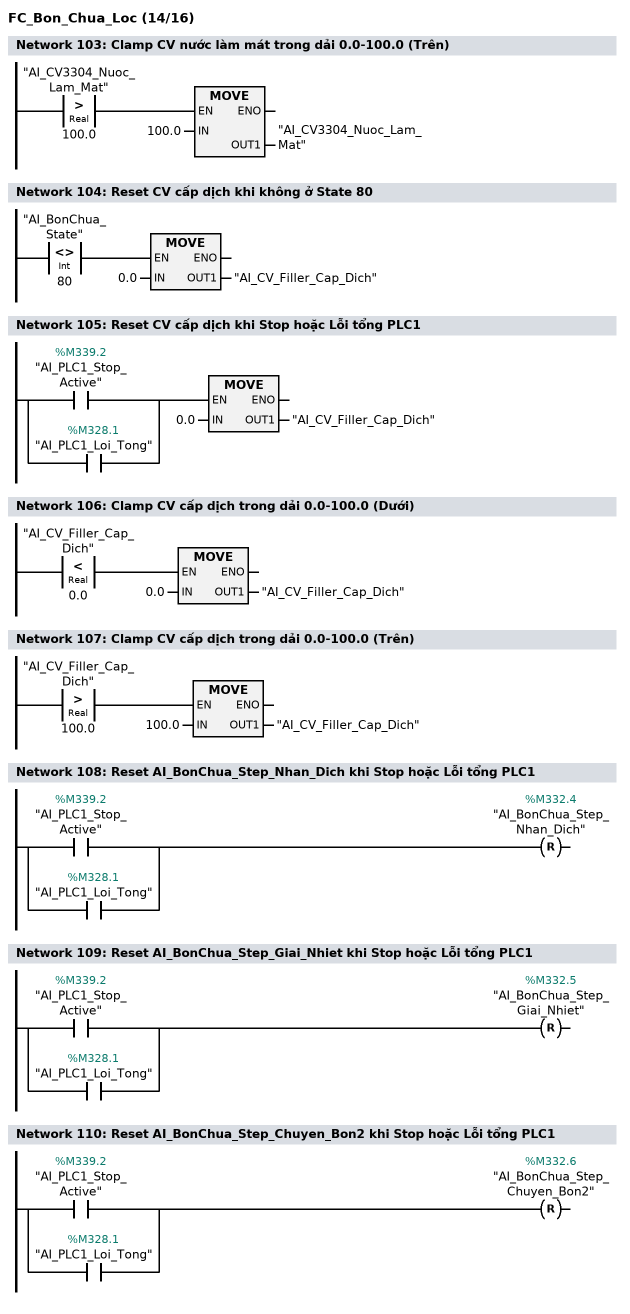
   RUNG wire#powerrail
      { S7_Templates := "SrcType := Real" } GT_Contact(in1 := "AI_CV3304_Nuoc_Lam_Mat", in2 := 100.0)
      { S7_GenerateENO := "TRUE" } Move(in := 100.0, out1 => "AI_CV3304_Nuoc_Lam_Mat")
   END_RUNG
   // the same network as SCL:
   IF "AI_CV3304_Nuoc_Lam_Mat" > 100.0 THEN "AI_CV3304_Nuoc_Lam_Mat" := 100.0; END_IF;
END_REGION

REGION Network 104: Reset CV cấp dịch khi không ở State 80
   RUNG wire#powerrail
      { S7_Templates := "SrcType := Int" } NE_Contact(in1 := "AI_BonChua_State", in2 := 80)
      { S7_GenerateENO := "TRUE" } Move(in := 0.0, out1 => "AI_CV_Filler_Cap_Dich")
   END_RUNG
   // the same network as SCL:
   IF "AI_BonChua_State" <> 80 THEN "AI_CV_Filler_Cap_Dich" := 0.0; END_IF;
END_REGION

REGION Network 105: Reset CV cấp dịch khi Stop hoặc Lỗi tổng PLC1
   RUNG wire#powerrail
      Contact( "AI_PLC1_Stop_Active" )
      wire#w1
      { S7_GenerateENO := "TRUE" } Move(in := 0.0, out1 => "AI_CV_Filler_Cap_Dich")
   END_RUNG
   RUNG wire#powerrail
      Contact( "AI_PLC1_Loi_Tong" )
   END_RUNG wire#w1
   // the same network as SCL:
   IF "AI_PLC1_Stop_Active" OR "AI_PLC1_Loi_Tong" THEN "AI_CV_Filler_Cap_Dich" := 0.0; END_IF;
END_REGION

REGION Network 106: Clamp CV cấp dịch trong dải 0.0-100.0 (Dưới)
   RUNG wire#powerrail
      { S7_Templates := "SrcType := Real" } LT_Contact(in1 := "AI_CV_Filler_Cap_Dich", in2 := 0.0)
      { S7_GenerateENO := "TRUE" } Move(in := 0.0, out1 => "AI_CV_Filler_Cap_Dich")
   END_RUNG
   // the same network as SCL:
   IF "AI_CV_Filler_Cap_Dich" < 0.0 THEN "AI_CV_Filler_Cap_Dich" := 0.0; END_IF;
END_REGION

REGION Network 107: Clamp CV cấp dịch trong dải 0.0-100.0 (Trên)
   RUNG wire#powerrail
      { S7_Templates := "SrcType := Real" } GT_Contact(in1 := "AI_CV_Filler_Cap_Dich", in2 := 100.0)
      { S7_GenerateENO := "TRUE" } Move(in := 100.0, out1 => "AI_CV_Filler_Cap_Dich")
   END_RUNG
   // the same network as SCL:
   IF "AI_CV_Filler_Cap_Dich" > 100.0 THEN "AI_CV_Filler_Cap_Dich" := 100.0; END_IF;
END_REGION

REGION Network 108: Reset AI_BonChua_Step_Nhan_Dich khi Stop hoặc Lỗi tổng PLC1
   RUNG wire#powerrail
      Contact( "AI_PLC1_Stop_Active" )
      wire#w1
      R_Coil( "AI_BonChua_Step_Nhan_Dich" )
   END_RUNG
   RUNG wire#powerrail
      Contact( "AI_PLC1_Loi_Tong" )
   END_RUNG wire#w1
   // the same network as SCL:
   IF "AI_PLC1_Stop_Active" OR "AI_PLC1_Loi_Tong" THEN "AI_BonChua_Step_Nhan_Dich" := FALSE; END_IF;
END_REGION

REGION Network 109: Reset AI_BonChua_Step_Giai_Nhiet khi Stop hoặc Lỗi tổng PLC1
   RUNG wire#powerrail
      Contact( "AI_PLC1_Stop_Active" )
      wire#w1
      R_Coil( "AI_BonChua_Step_Giai_Nhiet" )
   END_RUNG
   RUNG wire#powerrail
      Contact( "AI_PLC1_Loi_Tong" )
   END_RUNG wire#w1
   // the same network as SCL:
   IF "AI_PLC1_Stop_Active" OR "AI_PLC1_Loi_Tong" THEN "AI_BonChua_Step_Giai_Nhiet" := FALSE; END_IF;
END_REGION

REGION Network 110: Reset AI_BonChua_Step_Chuyen_Bon2 khi Stop hoặc Lỗi tổng PLC1
   RUNG wire#powerrail
      Contact( "AI_PLC1_Stop_Active" )
      wire#w1
      R_Coil( "AI_BonChua_Step_Chuyen_Bon2" )
   END_RUNG
   RUNG wire#powerrail
      Contact( "AI_PLC1_Loi_Tong" )
   END_RUNG wire#w1
   // the same network as SCL:
   IF "AI_PLC1_Stop_Active" OR "AI_PLC1_Loi_Tong" THEN "AI_BonChua_Step_Chuyen_Bon2" := FALSE; END_IF;
END_REGION

REGION Network 111: Reset AI_BonChua_Step_Loc_Chiet khi Stop hoặc Lỗi tổng PLC1
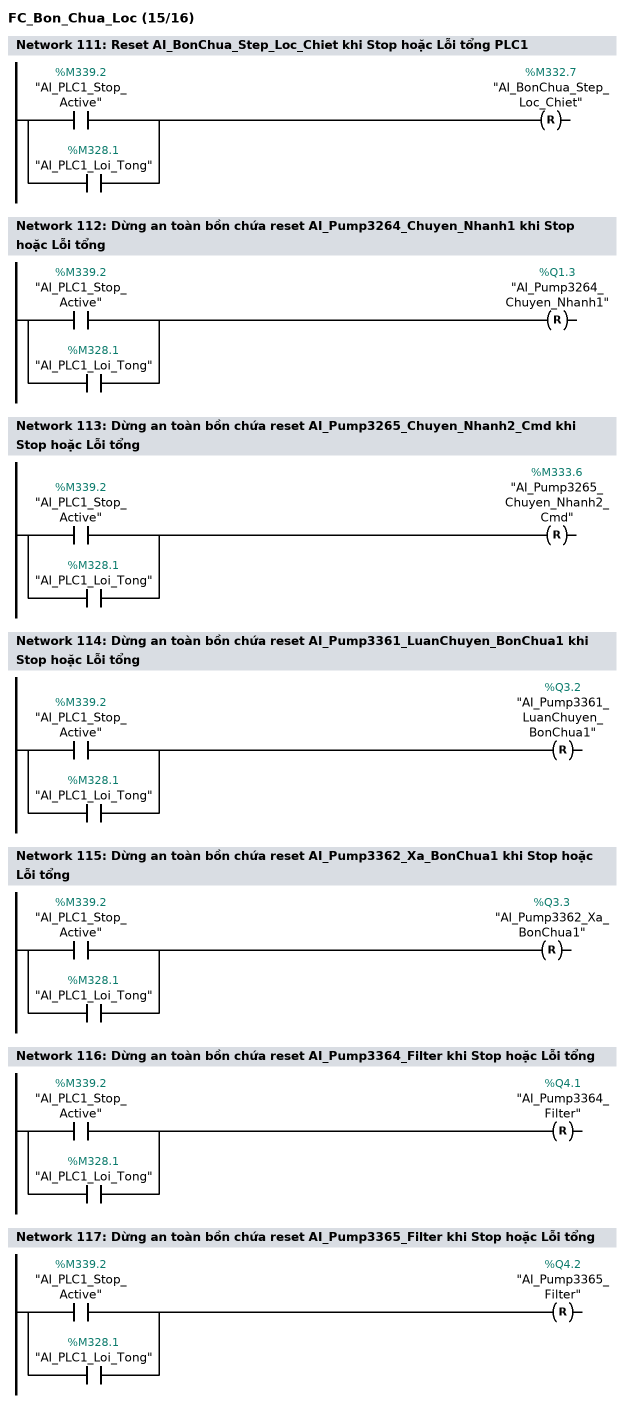
   RUNG wire#powerrail
      Contact( "AI_PLC1_Stop_Active" )
      wire#w1
      R_Coil( "AI_BonChua_Step_Loc_Chiet" )
   END_RUNG
   RUNG wire#powerrail
      Contact( "AI_PLC1_Loi_Tong" )
   END_RUNG wire#w1
   // the same network as SCL:
   IF "AI_PLC1_Stop_Active" OR "AI_PLC1_Loi_Tong" THEN "AI_BonChua_Step_Loc_Chiet" := FALSE; END_IF;
END_REGION

REGION Network 112: Dừng an toàn bồn chứa reset AI_Pump3264_Chuyen_Nhanh1 khi Stop hoặc Lỗi tổng
   RUNG wire#powerrail
      Contact( "AI_PLC1_Stop_Active" )
      wire#w1
      R_Coil( "AI_Pump3264_Chuyen_Nhanh1" )
   END_RUNG
   RUNG wire#powerrail
      Contact( "AI_PLC1_Loi_Tong" )
   END_RUNG wire#w1
   // the same network as SCL:
   IF "AI_PLC1_Stop_Active" OR "AI_PLC1_Loi_Tong" THEN "AI_Pump3264_Chuyen_Nhanh1" := FALSE; END_IF;
END_REGION

REGION Network 113: Dừng an toàn bồn chứa reset AI_Pump3265_Chuyen_Nhanh2_Cmd khi Stop hoặc Lỗi tổng
   RUNG wire#powerrail
      Contact( "AI_PLC1_Stop_Active" )
      wire#w1
      R_Coil( "AI_Pump3265_Chuyen_Nhanh2_Cmd" )
   END_RUNG
   RUNG wire#powerrail
      Contact( "AI_PLC1_Loi_Tong" )
   END_RUNG wire#w1
   // the same network as SCL:
   IF "AI_PLC1_Stop_Active" OR "AI_PLC1_Loi_Tong" THEN "AI_Pump3265_Chuyen_Nhanh2_Cmd" := FALSE; END_IF;
END_REGION

REGION Network 114: Dừng an toàn bồn chứa reset AI_Pump3361_LuanChuyen_BonChua1 khi Stop hoặc Lỗi tổng
   RUNG wire#powerrail
      Contact( "AI_PLC1_Stop_Active" )
      wire#w1
      R_Coil( "AI_Pump3361_LuanChuyen_BonChua1" )
   END_RUNG
   RUNG wire#powerrail
      Contact( "AI_PLC1_Loi_Tong" )
   END_RUNG wire#w1
   // the same network as SCL:
   IF "AI_PLC1_Stop_Active" OR "AI_PLC1_Loi_Tong" THEN "AI_Pump3361_LuanChuyen_BonChua1" := FALSE; END_IF;
END_REGION

REGION Network 115: Dừng an toàn bồn chứa reset AI_Pump3362_Xa_BonChua1 khi Stop hoặc Lỗi tổng
   RUNG wire#powerrail
      Contact( "AI_PLC1_Stop_Active" )
      wire#w1
      R_Coil( "AI_Pump3362_Xa_BonChua1" )
   END_RUNG
   RUNG wire#powerrail
      Contact( "AI_PLC1_Loi_Tong" )
   END_RUNG wire#w1
   // the same network as SCL:
   IF "AI_PLC1_Stop_Active" OR "AI_PLC1_Loi_Tong" THEN "AI_Pump3362_Xa_BonChua1" := FALSE; END_IF;
END_REGION

REGION Network 116: Dừng an toàn bồn chứa reset AI_Pump3364_Filter khi Stop hoặc Lỗi tổng
   RUNG wire#powerrail
      Contact( "AI_PLC1_Stop_Active" )
      wire#w1
      R_Coil( "AI_Pump3364_Filter" )
   END_RUNG
   RUNG wire#powerrail
      Contact( "AI_PLC1_Loi_Tong" )
   END_RUNG wire#w1
   // the same network as SCL:
   IF "AI_PLC1_Stop_Active" OR "AI_PLC1_Loi_Tong" THEN "AI_Pump3364_Filter" := FALSE; END_IF;
END_REGION

REGION Network 117: Dừng an toàn bồn chứa reset AI_Pump3365_Filter khi Stop hoặc Lỗi tổng
   RUNG wire#powerrail
      Contact( "AI_PLC1_Stop_Active" )
      wire#w1
      R_Coil( "AI_Pump3365_Filter" )
   END_RUNG
   RUNG wire#powerrail
      Contact( "AI_PLC1_Loi_Tong" )
   END_RUNG wire#w1
   // the same network as SCL:
   IF "AI_PLC1_Stop_Active" OR "AI_PLC1_Loi_Tong" THEN "AI_Pump3365_Filter" := FALSE; END_IF;
END_REGION

REGION Network 118: Dừng an toàn bồn chứa reset AI_V3331_Xa_BonChua1 khi Stop hoặc Lỗi tổng
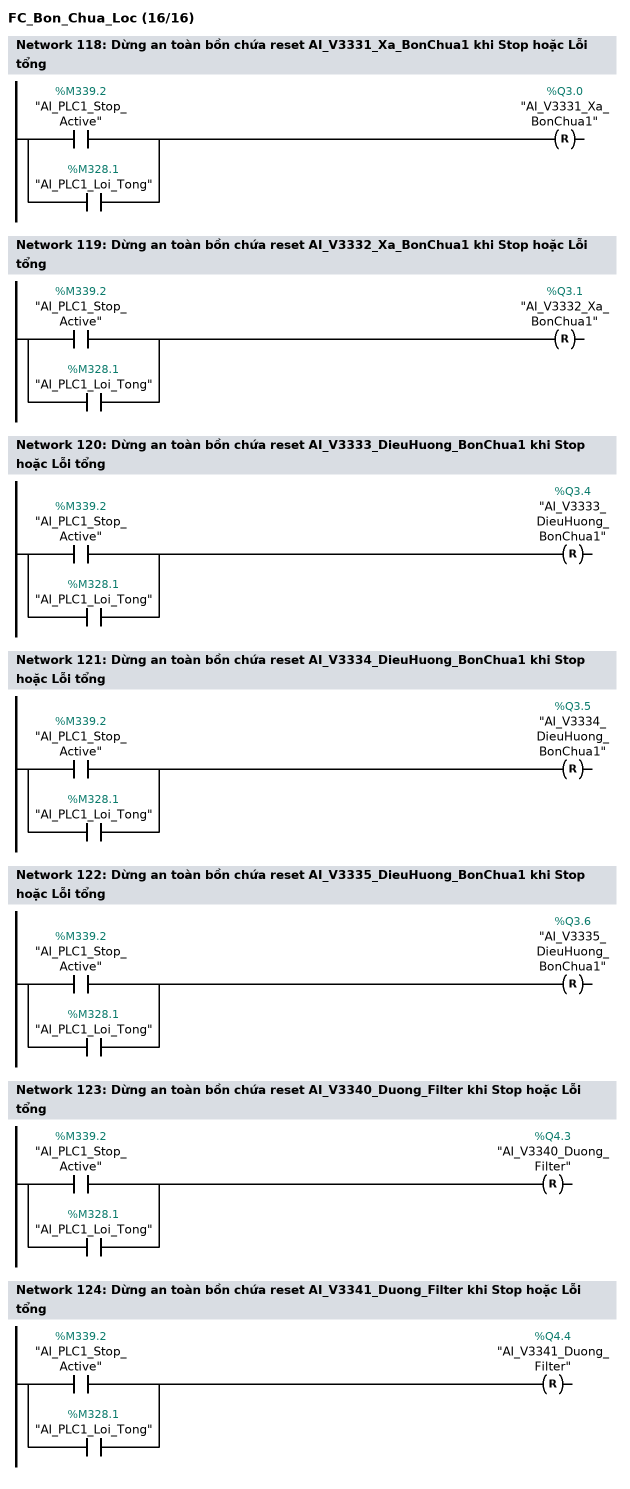
   RUNG wire#powerrail
      Contact( "AI_PLC1_Stop_Active" )
      wire#w1
      R_Coil( "AI_V3331_Xa_BonChua1" )
   END_RUNG
   RUNG wire#powerrail
      Contact( "AI_PLC1_Loi_Tong" )
   END_RUNG wire#w1
   // the same network as SCL:
   IF "AI_PLC1_Stop_Active" OR "AI_PLC1_Loi_Tong" THEN "AI_V3331_Xa_BonChua1" := FALSE; END_IF;
END_REGION

REGION Network 119: Dừng an toàn bồn chứa reset AI_V3332_Xa_BonChua1 khi Stop hoặc Lỗi tổng
   RUNG wire#powerrail
      Contact( "AI_PLC1_Stop_Active" )
      wire#w1
      R_Coil( "AI_V3332_Xa_BonChua1" )
   END_RUNG
   RUNG wire#powerrail
      Contact( "AI_PLC1_Loi_Tong" )
   END_RUNG wire#w1
   // the same network as SCL:
   IF "AI_PLC1_Stop_Active" OR "AI_PLC1_Loi_Tong" THEN "AI_V3332_Xa_BonChua1" := FALSE; END_IF;
END_REGION

REGION Network 120: Dừng an toàn bồn chứa reset AI_V3333_DieuHuong_BonChua1 khi Stop hoặc Lỗi tổng
   RUNG wire#powerrail
      Contact( "AI_PLC1_Stop_Active" )
      wire#w1
      R_Coil( "AI_V3333_DieuHuong_BonChua1" )
   END_RUNG
   RUNG wire#powerrail
      Contact( "AI_PLC1_Loi_Tong" )
   END_RUNG wire#w1
   // the same network as SCL:
   IF "AI_PLC1_Stop_Active" OR "AI_PLC1_Loi_Tong" THEN "AI_V3333_DieuHuong_BonChua1" := FALSE; END_IF;
END_REGION

REGION Network 121: Dừng an toàn bồn chứa reset AI_V3334_DieuHuong_BonChua1 khi Stop hoặc Lỗi tổng
   RUNG wire#powerrail
      Contact( "AI_PLC1_Stop_Active" )
      wire#w1
      R_Coil( "AI_V3334_DieuHuong_BonChua1" )
   END_RUNG
   RUNG wire#powerrail
      Contact( "AI_PLC1_Loi_Tong" )
   END_RUNG wire#w1
   // the same network as SCL:
   IF "AI_PLC1_Stop_Active" OR "AI_PLC1_Loi_Tong" THEN "AI_V3334_DieuHuong_BonChua1" := FALSE; END_IF;
END_REGION

REGION Network 122: Dừng an toàn bồn chứa reset AI_V3335_DieuHuong_BonChua1 khi Stop hoặc Lỗi tổng
   RUNG wire#powerrail
      Contact( "AI_PLC1_Stop_Active" )
      wire#w1
      R_Coil( "AI_V3335_DieuHuong_BonChua1" )
   END_RUNG
   RUNG wire#powerrail
      Contact( "AI_PLC1_Loi_Tong" )
   END_RUNG wire#w1
   // the same network as SCL:
   IF "AI_PLC1_Stop_Active" OR "AI_PLC1_Loi_Tong" THEN "AI_V3335_DieuHuong_BonChua1" := FALSE; END_IF;
END_REGION

REGION Network 123: Dừng an toàn bồn chứa reset AI_V3340_Duong_Filter khi Stop hoặc Lỗi tổng
   RUNG wire#powerrail
      Contact( "AI_PLC1_Stop_Active" )
      wire#w1
      R_Coil( "AI_V3340_Duong_Filter" )
   END_RUNG
   RUNG wire#powerrail
      Contact( "AI_PLC1_Loi_Tong" )
   END_RUNG wire#w1
   // the same network as SCL:
   IF "AI_PLC1_Stop_Active" OR "AI_PLC1_Loi_Tong" THEN "AI_V3340_Duong_Filter" := FALSE; END_IF;
END_REGION

REGION Network 124: Dừng an toàn bồn chứa reset AI_V3341_Duong_Filter khi Stop hoặc Lỗi tổng
   RUNG wire#powerrail
      Contact( "AI_PLC1_Stop_Active" )
      wire#w1
      R_Coil( "AI_V3341_Duong_Filter" )
   END_RUNG
   RUNG wire#powerrail
      Contact( "AI_PLC1_Loi_Tong" )
   END_RUNG wire#w1
   // the same network as SCL:
   IF "AI_PLC1_Stop_Active" OR "AI_PLC1_Loi_Tong" THEN "AI_V3341_Duong_Filter" := FALSE; END_IF;
END_REGION
END_FUNCTION

FUNCTION "FC_HMI_Mirror_PLC1" : Void   // FC40, LAD
{ S7_Optimized_Access := 'TRUE' }
VERSION : 0.1
// stored: AutoNumber true, IsIECCheckEnabled false
BEGIN

REGION Network 1: Mirror AI_V3230_Nuoc_Bon1
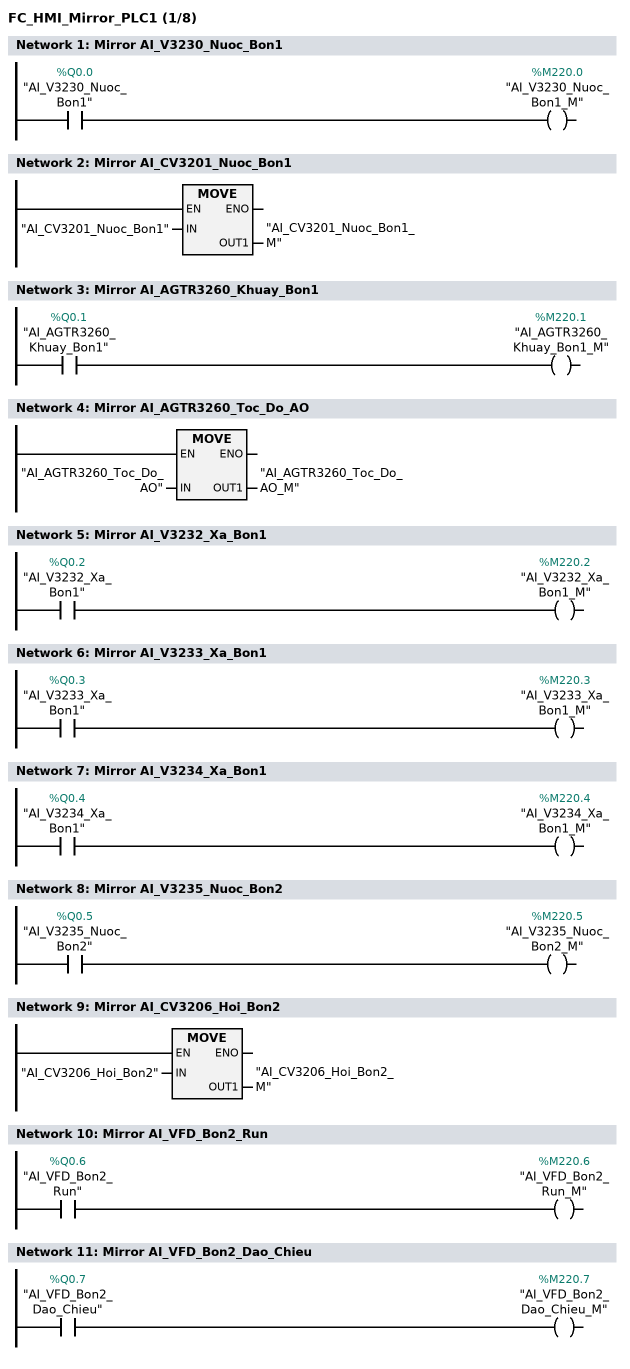
   RUNG wire#powerrail
      Contact( "AI_V3230_Nuoc_Bon1" )
      Coil( "AI_V3230_Nuoc_Bon1_M" )
   END_RUNG
   // the same network as SCL:
   "AI_V3230_Nuoc_Bon1_M" := "AI_V3230_Nuoc_Bon1";
END_REGION

REGION Network 2: Mirror AI_CV3201_Nuoc_Bon1
   RUNG wire#powerrail
      { S7_GenerateENO := "TRUE" } Move(in := "AI_CV3201_Nuoc_Bon1", out1 => "AI_CV3201_Nuoc_Bon1_M")
   END_RUNG
   // the same network as SCL:
   "AI_CV3201_Nuoc_Bon1_M" := "AI_CV3201_Nuoc_Bon1";
END_REGION

REGION Network 3: Mirror AI_AGTR3260_Khuay_Bon1
   RUNG wire#powerrail
      Contact( "AI_AGTR3260_Khuay_Bon1" )
      Coil( "AI_AGTR3260_Khuay_Bon1_M" )
   END_RUNG
   // the same network as SCL:
   "AI_AGTR3260_Khuay_Bon1_M" := "AI_AGTR3260_Khuay_Bon1";
END_REGION

REGION Network 4: Mirror AI_AGTR3260_Toc_Do_AO
   RUNG wire#powerrail
      { S7_GenerateENO := "TRUE" } Move(in := "AI_AGTR3260_Toc_Do_AO", out1 => "AI_AGTR3260_Toc_Do_AO_M")
   END_RUNG
   // the same network as SCL:
   "AI_AGTR3260_Toc_Do_AO_M" := "AI_AGTR3260_Toc_Do_AO";
END_REGION

REGION Network 5: Mirror AI_V3232_Xa_Bon1
   RUNG wire#powerrail
      Contact( "AI_V3232_Xa_Bon1" )
      Coil( "AI_V3232_Xa_Bon1_M" )
   END_RUNG
   // the same network as SCL:
   "AI_V3232_Xa_Bon1_M" := "AI_V3232_Xa_Bon1";
END_REGION

REGION Network 6: Mirror AI_V3233_Xa_Bon1
   RUNG wire#powerrail
      Contact( "AI_V3233_Xa_Bon1" )
      Coil( "AI_V3233_Xa_Bon1_M" )
   END_RUNG
   // the same network as SCL:
   "AI_V3233_Xa_Bon1_M" := "AI_V3233_Xa_Bon1";
END_REGION

REGION Network 7: Mirror AI_V3234_Xa_Bon1
   RUNG wire#powerrail
      Contact( "AI_V3234_Xa_Bon1" )
      Coil( "AI_V3234_Xa_Bon1_M" )
   END_RUNG
   // the same network as SCL:
   "AI_V3234_Xa_Bon1_M" := "AI_V3234_Xa_Bon1";
END_REGION

REGION Network 8: Mirror AI_V3235_Nuoc_Bon2
   RUNG wire#powerrail
      Contact( "AI_V3235_Nuoc_Bon2" )
      Coil( "AI_V3235_Nuoc_Bon2_M" )
   END_RUNG
   // the same network as SCL:
   "AI_V3235_Nuoc_Bon2_M" := "AI_V3235_Nuoc_Bon2";
END_REGION

REGION Network 9: Mirror AI_CV3206_Hoi_Bon2
   RUNG wire#powerrail
      { S7_GenerateENO := "TRUE" } Move(in := "AI_CV3206_Hoi_Bon2", out1 => "AI_CV3206_Hoi_Bon2_M")
   END_RUNG
   // the same network as SCL:
   "AI_CV3206_Hoi_Bon2_M" := "AI_CV3206_Hoi_Bon2";
END_REGION

REGION Network 10: Mirror AI_VFD_Bon2_Run
   RUNG wire#powerrail
      Contact( "AI_VFD_Bon2_Run" )
      Coil( "AI_VFD_Bon2_Run_M" )
   END_RUNG
   // the same network as SCL:
   "AI_VFD_Bon2_Run_M" := "AI_VFD_Bon2_Run";
END_REGION

REGION Network 11: Mirror AI_VFD_Bon2_Dao_Chieu
   RUNG wire#powerrail
      Contact( "AI_VFD_Bon2_Dao_Chieu" )
      Coil( "AI_VFD_Bon2_Dao_Chieu_M" )
   END_RUNG
   // the same network as SCL:
   "AI_VFD_Bon2_Dao_Chieu_M" := "AI_VFD_Bon2_Dao_Chieu";
END_REGION

REGION Network 12: Mirror AI_VFD_Bon2_Toc_Do_AO
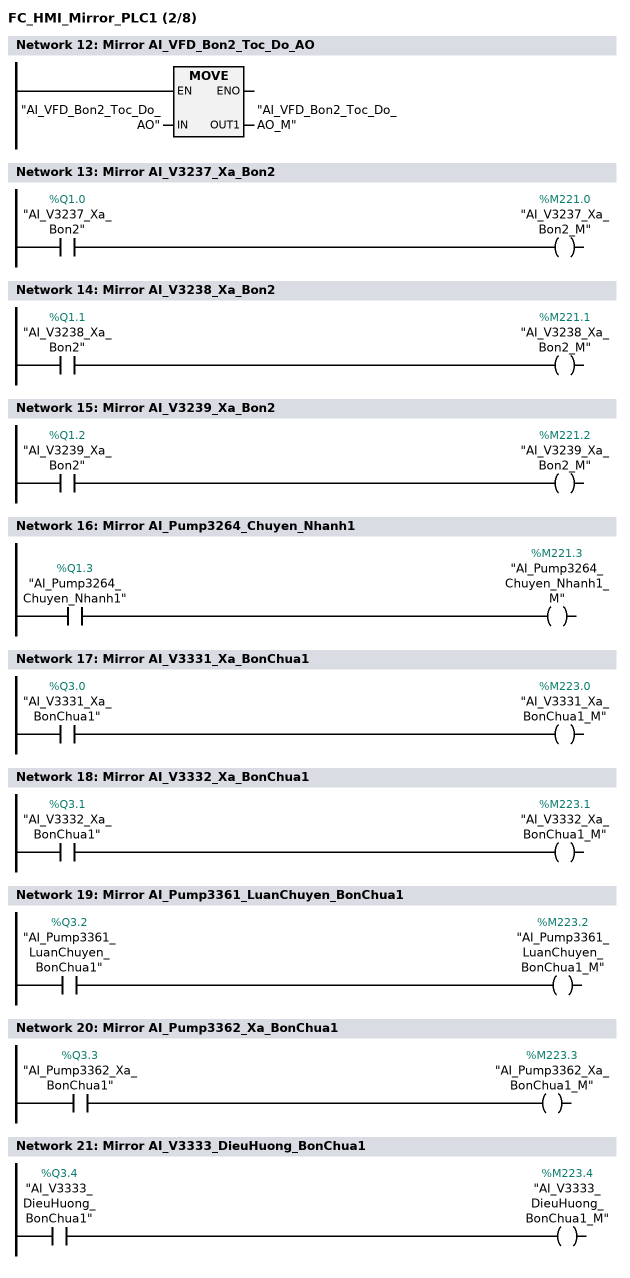
   RUNG wire#powerrail
      { S7_GenerateENO := "TRUE" } Move(in := "AI_VFD_Bon2_Toc_Do_AO", out1 => "AI_VFD_Bon2_Toc_Do_AO_M")
   END_RUNG
   // the same network as SCL:
   "AI_VFD_Bon2_Toc_Do_AO_M" := "AI_VFD_Bon2_Toc_Do_AO";
END_REGION

REGION Network 13: Mirror AI_V3237_Xa_Bon2
   RUNG wire#powerrail
      Contact( "AI_V3237_Xa_Bon2" )
      Coil( "AI_V3237_Xa_Bon2_M" )
   END_RUNG
   // the same network as SCL:
   "AI_V3237_Xa_Bon2_M" := "AI_V3237_Xa_Bon2";
END_REGION

REGION Network 14: Mirror AI_V3238_Xa_Bon2
   RUNG wire#powerrail
      Contact( "AI_V3238_Xa_Bon2" )
      Coil( "AI_V3238_Xa_Bon2_M" )
   END_RUNG
   // the same network as SCL:
   "AI_V3238_Xa_Bon2_M" := "AI_V3238_Xa_Bon2";
END_REGION

REGION Network 15: Mirror AI_V3239_Xa_Bon2
   RUNG wire#powerrail
      Contact( "AI_V3239_Xa_Bon2" )
      Coil( "AI_V3239_Xa_Bon2_M" )
   END_RUNG
   // the same network as SCL:
   "AI_V3239_Xa_Bon2_M" := "AI_V3239_Xa_Bon2";
END_REGION

REGION Network 16: Mirror AI_Pump3264_Chuyen_Nhanh1
   RUNG wire#powerrail
      Contact( "AI_Pump3264_Chuyen_Nhanh1" )
      Coil( "AI_Pump3264_Chuyen_Nhanh1_M" )
   END_RUNG
   // the same network as SCL:
   "AI_Pump3264_Chuyen_Nhanh1_M" := "AI_Pump3264_Chuyen_Nhanh1";
END_REGION

REGION Network 17: Mirror AI_V3331_Xa_BonChua1
   RUNG wire#powerrail
      Contact( "AI_V3331_Xa_BonChua1" )
      Coil( "AI_V3331_Xa_BonChua1_M" )
   END_RUNG
   // the same network as SCL:
   "AI_V3331_Xa_BonChua1_M" := "AI_V3331_Xa_BonChua1";
END_REGION

REGION Network 18: Mirror AI_V3332_Xa_BonChua1
   RUNG wire#powerrail
      Contact( "AI_V3332_Xa_BonChua1" )
      Coil( "AI_V3332_Xa_BonChua1_M" )
   END_RUNG
   // the same network as SCL:
   "AI_V3332_Xa_BonChua1_M" := "AI_V3332_Xa_BonChua1";
END_REGION

REGION Network 19: Mirror AI_Pump3361_LuanChuyen_BonChua1
   RUNG wire#powerrail
      Contact( "AI_Pump3361_LuanChuyen_BonChua1" )
      Coil( "AI_Pump3361_LuanChuyen_BonChua1_M" )
   END_RUNG
   // the same network as SCL:
   "AI_Pump3361_LuanChuyen_BonChua1_M" := "AI_Pump3361_LuanChuyen_BonChua1";
END_REGION

REGION Network 20: Mirror AI_Pump3362_Xa_BonChua1
   RUNG wire#powerrail
      Contact( "AI_Pump3362_Xa_BonChua1" )
      Coil( "AI_Pump3362_Xa_BonChua1_M" )
   END_RUNG
   // the same network as SCL:
   "AI_Pump3362_Xa_BonChua1_M" := "AI_Pump3362_Xa_BonChua1";
END_REGION

REGION Network 21: Mirror AI_V3333_DieuHuong_BonChua1
   RUNG wire#powerrail
      Contact( "AI_V3333_DieuHuong_BonChua1" )
      Coil( "AI_V3333_DieuHuong_BonChua1_M" )
   END_RUNG
   // the same network as SCL:
   "AI_V3333_DieuHuong_BonChua1_M" := "AI_V3333_DieuHuong_BonChua1";
END_REGION

REGION Network 22: Mirror AI_V3334_DieuHuong_BonChua1
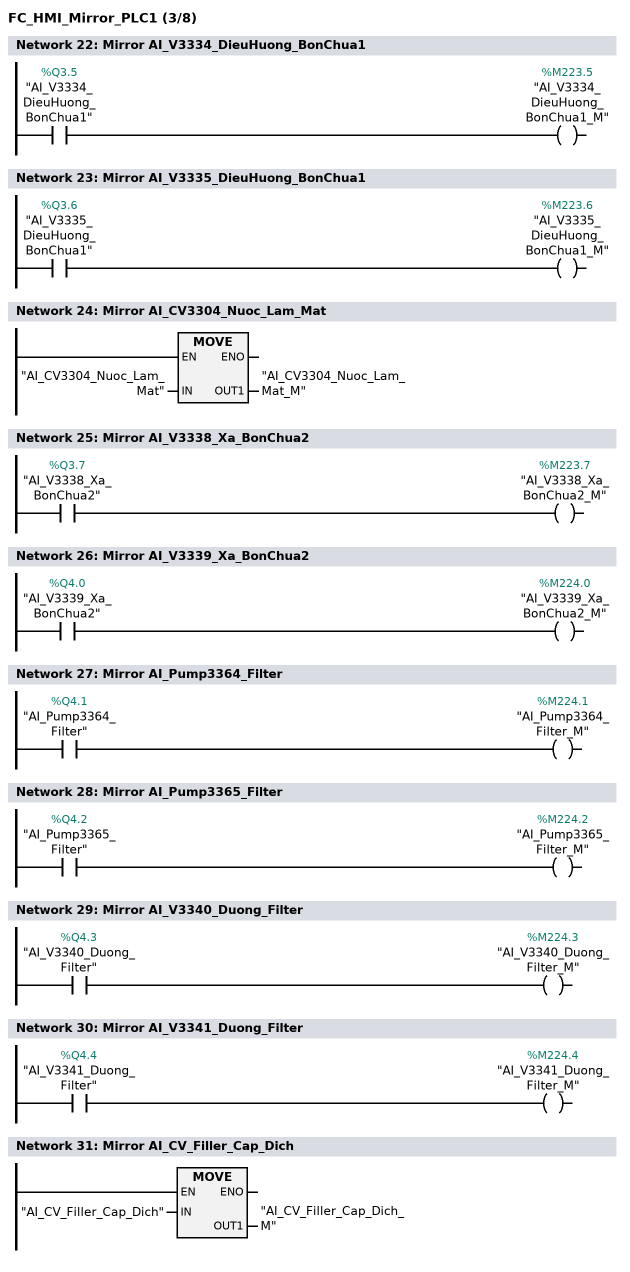
   RUNG wire#powerrail
      Contact( "AI_V3334_DieuHuong_BonChua1" )
      Coil( "AI_V3334_DieuHuong_BonChua1_M" )
   END_RUNG
   // the same network as SCL:
   "AI_V3334_DieuHuong_BonChua1_M" := "AI_V3334_DieuHuong_BonChua1";
END_REGION

REGION Network 23: Mirror AI_V3335_DieuHuong_BonChua1
   RUNG wire#powerrail
      Contact( "AI_V3335_DieuHuong_BonChua1" )
      Coil( "AI_V3335_DieuHuong_BonChua1_M" )
   END_RUNG
   // the same network as SCL:
   "AI_V3335_DieuHuong_BonChua1_M" := "AI_V3335_DieuHuong_BonChua1";
END_REGION

REGION Network 24: Mirror AI_CV3304_Nuoc_Lam_Mat
   RUNG wire#powerrail
      { S7_GenerateENO := "TRUE" } Move(in := "AI_CV3304_Nuoc_Lam_Mat", out1 => "AI_CV3304_Nuoc_Lam_Mat_M")
   END_RUNG
   // the same network as SCL:
   "AI_CV3304_Nuoc_Lam_Mat_M" := "AI_CV3304_Nuoc_Lam_Mat";
END_REGION

REGION Network 25: Mirror AI_V3338_Xa_BonChua2
   RUNG wire#powerrail
      Contact( "AI_V3338_Xa_BonChua2" )
      Coil( "AI_V3338_Xa_BonChua2_M" )
   END_RUNG
   // the same network as SCL:
   "AI_V3338_Xa_BonChua2_M" := "AI_V3338_Xa_BonChua2";
END_REGION

REGION Network 26: Mirror AI_V3339_Xa_BonChua2
   RUNG wire#powerrail
      Contact( "AI_V3339_Xa_BonChua2" )
      Coil( "AI_V3339_Xa_BonChua2_M" )
   END_RUNG
   // the same network as SCL:
   "AI_V3339_Xa_BonChua2_M" := "AI_V3339_Xa_BonChua2";
END_REGION

REGION Network 27: Mirror AI_Pump3364_Filter
   RUNG wire#powerrail
      Contact( "AI_Pump3364_Filter" )
      Coil( "AI_Pump3364_Filter_M" )
   END_RUNG
   // the same network as SCL:
   "AI_Pump3364_Filter_M" := "AI_Pump3364_Filter";
END_REGION

REGION Network 28: Mirror AI_Pump3365_Filter
   RUNG wire#powerrail
      Contact( "AI_Pump3365_Filter" )
      Coil( "AI_Pump3365_Filter_M" )
   END_RUNG
   // the same network as SCL:
   "AI_Pump3365_Filter_M" := "AI_Pump3365_Filter";
END_REGION

REGION Network 29: Mirror AI_V3340_Duong_Filter
   RUNG wire#powerrail
      Contact( "AI_V3340_Duong_Filter" )
      Coil( "AI_V3340_Duong_Filter_M" )
   END_RUNG
   // the same network as SCL:
   "AI_V3340_Duong_Filter_M" := "AI_V3340_Duong_Filter";
END_REGION

REGION Network 30: Mirror AI_V3341_Duong_Filter
   RUNG wire#powerrail
      Contact( "AI_V3341_Duong_Filter" )
      Coil( "AI_V3341_Duong_Filter_M" )
   END_RUNG
   // the same network as SCL:
   "AI_V3341_Duong_Filter_M" := "AI_V3341_Duong_Filter";
END_REGION

REGION Network 31: Mirror AI_CV_Filler_Cap_Dich
   RUNG wire#powerrail
      { S7_GenerateENO := "TRUE" } Move(in := "AI_CV_Filler_Cap_Dich", out1 => "AI_CV_Filler_Cap_Dich_M")
   END_RUNG
   // the same network as SCL:
   "AI_CV_Filler_Cap_Dich_M" := "AI_CV_Filler_Cap_Dich";
END_REGION

REGION Network 32: Mirror AI_Coi_Bao_Dong
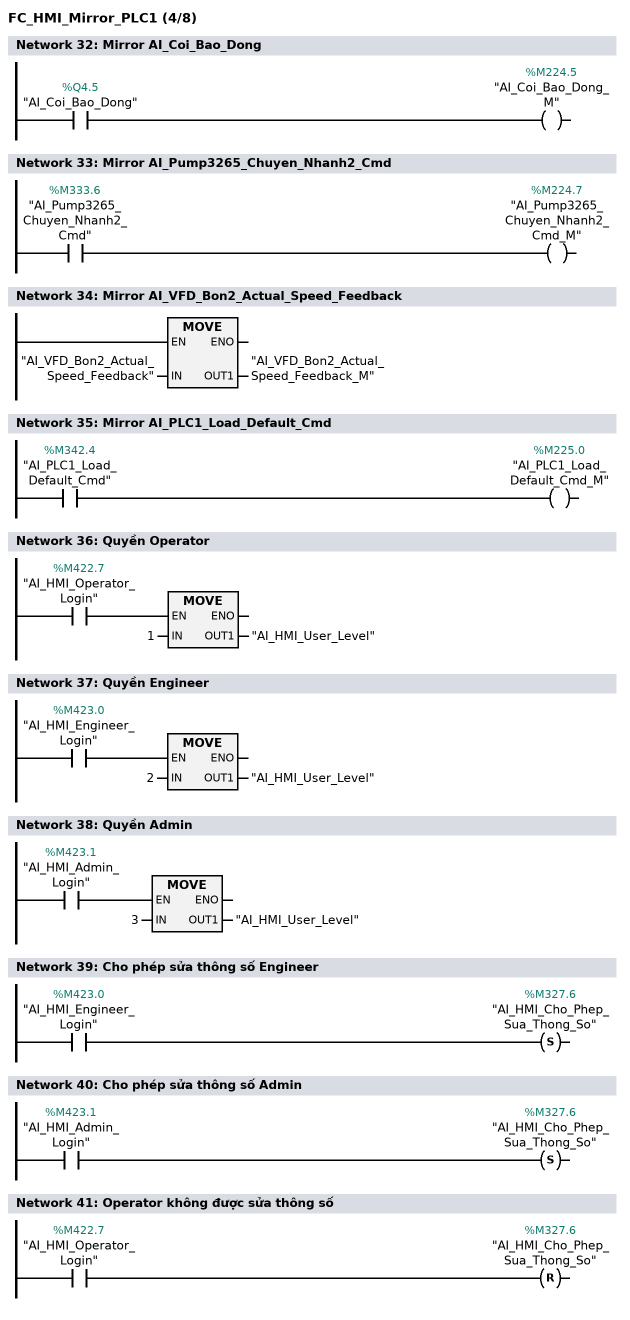
   RUNG wire#powerrail
      Contact( "AI_Coi_Bao_Dong" )
      Coil( "AI_Coi_Bao_Dong_M" )
   END_RUNG
   // the same network as SCL:
   "AI_Coi_Bao_Dong_M" := "AI_Coi_Bao_Dong";
END_REGION

REGION Network 33: Mirror AI_Pump3265_Chuyen_Nhanh2_Cmd
   RUNG wire#powerrail
      Contact( "AI_Pump3265_Chuyen_Nhanh2_Cmd" )
      Coil( "AI_Pump3265_Chuyen_Nhanh2_Cmd_M" )
   END_RUNG
   // the same network as SCL:
   "AI_Pump3265_Chuyen_Nhanh2_Cmd_M" := "AI_Pump3265_Chuyen_Nhanh2_Cmd";
END_REGION

REGION Network 34: Mirror AI_VFD_Bon2_Actual_Speed_Feedback
   RUNG wire#powerrail
      { S7_GenerateENO := "TRUE" } Move(in := "AI_VFD_Bon2_Actual_Speed_Feedback", out1 => "AI_VFD_Bon2_Actual_Speed_Feedback_M")
   END_RUNG
   // the same network as SCL:
   "AI_VFD_Bon2_Actual_Speed_Feedback_M" := "AI_VFD_Bon2_Actual_Speed_Feedback";
END_REGION

REGION Network 35: Mirror AI_PLC1_Load_Default_Cmd
   RUNG wire#powerrail
      Contact( "AI_PLC1_Load_Default_Cmd" )
      Coil( "AI_PLC1_Load_Default_Cmd_M" )
   END_RUNG
   // the same network as SCL:
   "AI_PLC1_Load_Default_Cmd_M" := "AI_PLC1_Load_Default_Cmd";
END_REGION

REGION Network 36: Quyền Operator
   RUNG wire#powerrail
      Contact( "AI_HMI_Operator_Login" )
      { S7_GenerateENO := "TRUE" } Move(in := 1, out1 => "AI_HMI_User_Level")
   END_RUNG
   // the same network as SCL:
   IF "AI_HMI_Operator_Login" THEN "AI_HMI_User_Level" := 1; END_IF;
END_REGION

REGION Network 37: Quyền Engineer
   RUNG wire#powerrail
      Contact( "AI_HMI_Engineer_Login" )
      { S7_GenerateENO := "TRUE" } Move(in := 2, out1 => "AI_HMI_User_Level")
   END_RUNG
   // the same network as SCL:
   IF "AI_HMI_Engineer_Login" THEN "AI_HMI_User_Level" := 2; END_IF;
END_REGION

REGION Network 38: Quyền Admin
   RUNG wire#powerrail
      Contact( "AI_HMI_Admin_Login" )
      { S7_GenerateENO := "TRUE" } Move(in := 3, out1 => "AI_HMI_User_Level")
   END_RUNG
   // the same network as SCL:
   IF "AI_HMI_Admin_Login" THEN "AI_HMI_User_Level" := 3; END_IF;
END_REGION

REGION Network 39: Cho phép sửa thông số Engineer
   RUNG wire#powerrail
      Contact( "AI_HMI_Engineer_Login" )
      S_Coil( "AI_HMI_Cho_Phep_Sua_Thong_So" )
   END_RUNG
   // the same network as SCL:
   IF "AI_HMI_Engineer_Login" THEN "AI_HMI_Cho_Phep_Sua_Thong_So" := TRUE; END_IF;
END_REGION

REGION Network 40: Cho phép sửa thông số Admin
   RUNG wire#powerrail
      Contact( "AI_HMI_Admin_Login" )
      S_Coil( "AI_HMI_Cho_Phep_Sua_Thong_So" )
   END_RUNG
   // the same network as SCL:
   IF "AI_HMI_Admin_Login" THEN "AI_HMI_Cho_Phep_Sua_Thong_So" := TRUE; END_IF;
END_REGION

REGION Network 41: Operator không được sửa thông số
   RUNG wire#powerrail
      Contact( "AI_HMI_Operator_Login" )
      R_Coil( "AI_HMI_Cho_Phep_Sua_Thong_So" )
   END_RUNG
   // the same network as SCL:
   IF "AI_HMI_Operator_Login" THEN "AI_HMI_Cho_Phep_Sua_Thong_So" := FALSE; END_IF;
END_REGION

REGION Network 42: Mã an toàn mặc định
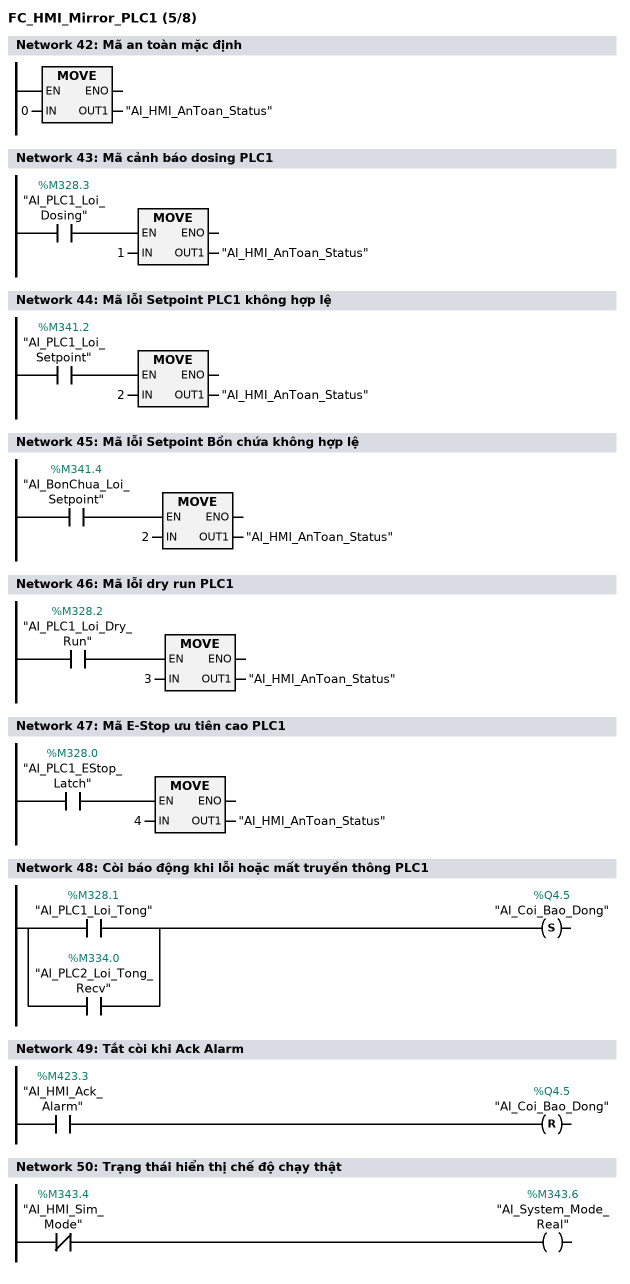
   RUNG wire#powerrail
      { S7_GenerateENO := "TRUE" } Move(in := 0, out1 => "AI_HMI_AnToan_Status")
   END_RUNG
   // the same network as SCL:
   "AI_HMI_AnToan_Status" := 0;
END_REGION

REGION Network 43: Mã cảnh báo dosing PLC1
   RUNG wire#powerrail
      Contact( "AI_PLC1_Loi_Dosing" )
      { S7_GenerateENO := "TRUE" } Move(in := 1, out1 => "AI_HMI_AnToan_Status")
   END_RUNG
   // the same network as SCL:
   IF "AI_PLC1_Loi_Dosing" THEN "AI_HMI_AnToan_Status" := 1; END_IF;
END_REGION

REGION Network 44: Mã lỗi Setpoint PLC1 không hợp lệ
   RUNG wire#powerrail
      Contact( "AI_PLC1_Loi_Setpoint" )
      { S7_GenerateENO := "TRUE" } Move(in := 2, out1 => "AI_HMI_AnToan_Status")
   END_RUNG
   // the same network as SCL:
   IF "AI_PLC1_Loi_Setpoint" THEN "AI_HMI_AnToan_Status" := 2; END_IF;
END_REGION

REGION Network 45: Mã lỗi Setpoint Bồn chứa không hợp lệ
   RUNG wire#powerrail
      Contact( "AI_BonChua_Loi_Setpoint" )
      { S7_GenerateENO := "TRUE" } Move(in := 2, out1 => "AI_HMI_AnToan_Status")
   END_RUNG
   // the same network as SCL:
   IF "AI_BonChua_Loi_Setpoint" THEN "AI_HMI_AnToan_Status" := 2; END_IF;
END_REGION

REGION Network 46: Mã lỗi dry run PLC1
   RUNG wire#powerrail
      Contact( "AI_PLC1_Loi_Dry_Run" )
      { S7_GenerateENO := "TRUE" } Move(in := 3, out1 => "AI_HMI_AnToan_Status")
   END_RUNG
   // the same network as SCL:
   IF "AI_PLC1_Loi_Dry_Run" THEN "AI_HMI_AnToan_Status" := 3; END_IF;
END_REGION

REGION Network 47: Mã E-Stop ưu tiên cao PLC1
   RUNG wire#powerrail
      Contact( "AI_PLC1_EStop_Latch" )
      { S7_GenerateENO := "TRUE" } Move(in := 4, out1 => "AI_HMI_AnToan_Status")
   END_RUNG
   // the same network as SCL:
   IF "AI_PLC1_EStop_Latch" THEN "AI_HMI_AnToan_Status" := 4; END_IF;
END_REGION

REGION Network 48: Còi báo động khi lỗi hoặc mất truyền thông PLC1
   RUNG wire#powerrail
      Contact( "AI_PLC1_Loi_Tong" )
      wire#w1
      S_Coil( "AI_Coi_Bao_Dong" )
   END_RUNG
   RUNG wire#powerrail
      Contact( "AI_PLC2_Loi_Tong_Recv" )
   END_RUNG wire#w1
   // the same network as SCL:
   IF "AI_PLC1_Loi_Tong" OR "AI_PLC2_Loi_Tong_Recv" THEN "AI_Coi_Bao_Dong" := TRUE; END_IF;
END_REGION

REGION Network 49: Tắt còi khi Ack Alarm
   RUNG wire#powerrail
      Contact( "AI_HMI_Ack_Alarm" )
      R_Coil( "AI_Coi_Bao_Dong" )
   END_RUNG
   // the same network as SCL:
   IF "AI_HMI_Ack_Alarm" THEN "AI_Coi_Bao_Dong" := FALSE; END_IF;
END_REGION

REGION Network 50: Trạng thái hiển thị chế độ chạy thật
   RUNG wire#powerrail
      I_Contact( "AI_HMI_Sim_Mode" )
      Coil( "AI_System_Mode_Real" )
   END_RUNG
   // the same network as SCL:
   "AI_System_Mode_Real" := NOT "AI_HMI_Sim_Mode";
END_REGION

REGION Network 51: Trạng thái hiển thị chế độ mô phỏng
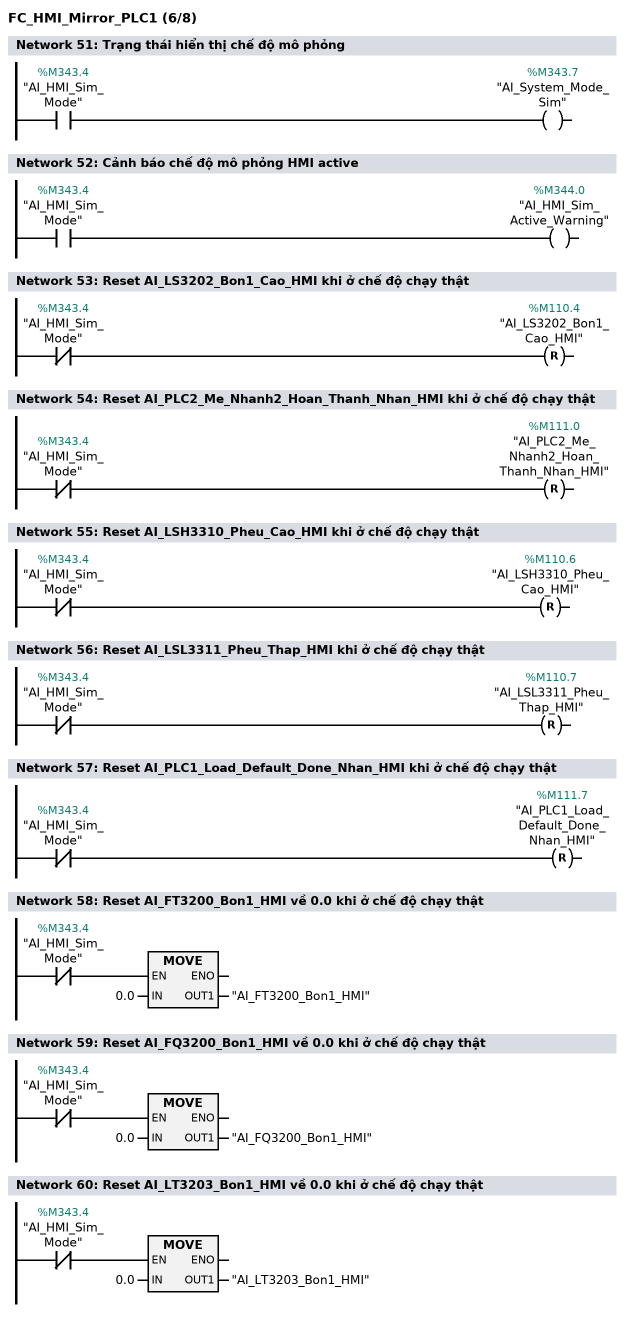
   RUNG wire#powerrail
      Contact( "AI_HMI_Sim_Mode" )
      Coil( "AI_System_Mode_Sim" )
   END_RUNG
   // the same network as SCL:
   "AI_System_Mode_Sim" := "AI_HMI_Sim_Mode";
END_REGION

REGION Network 52: Cảnh báo chế độ mô phỏng HMI active
   RUNG wire#powerrail
      Contact( "AI_HMI_Sim_Mode" )
      Coil( "AI_HMI_Sim_Active_Warning" )
   END_RUNG
   // the same network as SCL:
   "AI_HMI_Sim_Active_Warning" := "AI_HMI_Sim_Mode";
END_REGION

REGION Network 53: Reset AI_LS3202_Bon1_Cao_HMI khi ở chế độ chạy thật
   RUNG wire#powerrail
      I_Contact( "AI_HMI_Sim_Mode" )
      R_Coil( "AI_LS3202_Bon1_Cao_HMI" )
   END_RUNG
   // the same network as SCL:
   IF NOT "AI_HMI_Sim_Mode" THEN "AI_LS3202_Bon1_Cao_HMI" := FALSE; END_IF;
END_REGION

REGION Network 54: Reset AI_PLC2_Me_Nhanh2_Hoan_Thanh_Nhan_HMI khi ở chế độ chạy thật
   RUNG wire#powerrail
      I_Contact( "AI_HMI_Sim_Mode" )
      R_Coil( "AI_PLC2_Me_Nhanh2_Hoan_Thanh_Nhan_HMI" )
   END_RUNG
   // the same network as SCL:
   IF NOT "AI_HMI_Sim_Mode" THEN "AI_PLC2_Me_Nhanh2_Hoan_Thanh_Nhan_HMI" := FALSE; END_IF;
END_REGION

REGION Network 55: Reset AI_LSH3310_Pheu_Cao_HMI khi ở chế độ chạy thật
   RUNG wire#powerrail
      I_Contact( "AI_HMI_Sim_Mode" )
      R_Coil( "AI_LSH3310_Pheu_Cao_HMI" )
   END_RUNG
   // the same network as SCL:
   IF NOT "AI_HMI_Sim_Mode" THEN "AI_LSH3310_Pheu_Cao_HMI" := FALSE; END_IF;
END_REGION

REGION Network 56: Reset AI_LSL3311_Pheu_Thap_HMI khi ở chế độ chạy thật
   RUNG wire#powerrail
      I_Contact( "AI_HMI_Sim_Mode" )
      R_Coil( "AI_LSL3311_Pheu_Thap_HMI" )
   END_RUNG
   // the same network as SCL:
   IF NOT "AI_HMI_Sim_Mode" THEN "AI_LSL3311_Pheu_Thap_HMI" := FALSE; END_IF;
END_REGION

REGION Network 57: Reset AI_PLC1_Load_Default_Done_Nhan_HMI khi ở chế độ chạy thật
   RUNG wire#powerrail
      I_Contact( "AI_HMI_Sim_Mode" )
      R_Coil( "AI_PLC1_Load_Default_Done_Nhan_HMI" )
   END_RUNG
   // the same network as SCL:
   IF NOT "AI_HMI_Sim_Mode" THEN "AI_PLC1_Load_Default_Done_Nhan_HMI" := FALSE; END_IF;
END_REGION

REGION Network 58: Reset AI_FT3200_Bon1_HMI về 0.0 khi ở chế độ chạy thật
   RUNG wire#powerrail
      I_Contact( "AI_HMI_Sim_Mode" )
      { S7_GenerateENO := "TRUE" } Move(in := 0.0, out1 => "AI_FT3200_Bon1_HMI")
   END_RUNG
   // the same network as SCL:
   IF NOT "AI_HMI_Sim_Mode" THEN "AI_FT3200_Bon1_HMI" := 0.0; END_IF;
END_REGION

REGION Network 59: Reset AI_FQ3200_Bon1_HMI về 0.0 khi ở chế độ chạy thật
   RUNG wire#powerrail
      I_Contact( "AI_HMI_Sim_Mode" )
      { S7_GenerateENO := "TRUE" } Move(in := 0.0, out1 => "AI_FQ3200_Bon1_HMI")
   END_RUNG
   // the same network as SCL:
   IF NOT "AI_HMI_Sim_Mode" THEN "AI_FQ3200_Bon1_HMI" := 0.0; END_IF;
END_REGION

REGION Network 60: Reset AI_LT3203_Bon1_HMI về 0.0 khi ở chế độ chạy thật
   RUNG wire#powerrail
      I_Contact( "AI_HMI_Sim_Mode" )
      { S7_GenerateENO := "TRUE" } Move(in := 0.0, out1 => "AI_LT3203_Bon1_HMI")
   END_RUNG
   // the same network as SCL:
   IF NOT "AI_HMI_Sim_Mode" THEN "AI_LT3203_Bon1_HMI" := 0.0; END_IF;
END_REGION

REGION Network 61: Reset AI_TT3204_Bon1_HMI về 0.0 khi ở chế độ chạy thật
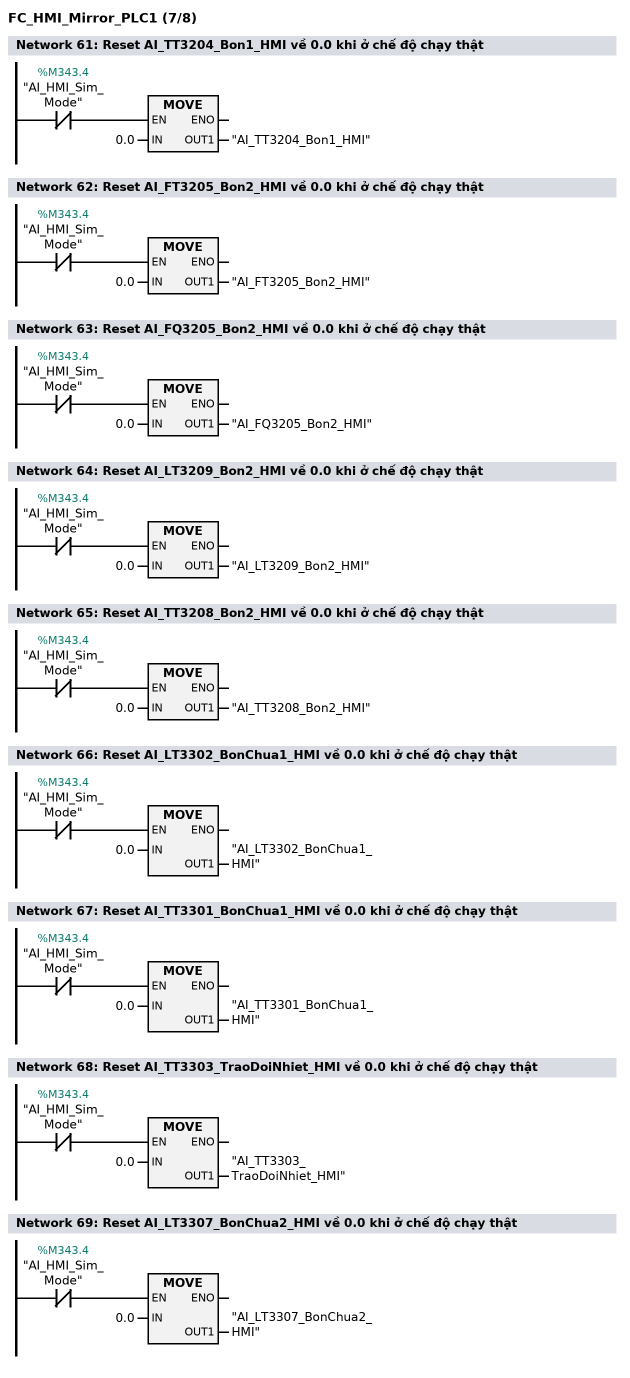
   RUNG wire#powerrail
      I_Contact( "AI_HMI_Sim_Mode" )
      { S7_GenerateENO := "TRUE" } Move(in := 0.0, out1 => "AI_TT3204_Bon1_HMI")
   END_RUNG
   // the same network as SCL:
   IF NOT "AI_HMI_Sim_Mode" THEN "AI_TT3204_Bon1_HMI" := 0.0; END_IF;
END_REGION

REGION Network 62: Reset AI_FT3205_Bon2_HMI về 0.0 khi ở chế độ chạy thật
   RUNG wire#powerrail
      I_Contact( "AI_HMI_Sim_Mode" )
      { S7_GenerateENO := "TRUE" } Move(in := 0.0, out1 => "AI_FT3205_Bon2_HMI")
   END_RUNG
   // the same network as SCL:
   IF NOT "AI_HMI_Sim_Mode" THEN "AI_FT3205_Bon2_HMI" := 0.0; END_IF;
END_REGION

REGION Network 63: Reset AI_FQ3205_Bon2_HMI về 0.0 khi ở chế độ chạy thật
   RUNG wire#powerrail
      I_Contact( "AI_HMI_Sim_Mode" )
      { S7_GenerateENO := "TRUE" } Move(in := 0.0, out1 => "AI_FQ3205_Bon2_HMI")
   END_RUNG
   // the same network as SCL:
   IF NOT "AI_HMI_Sim_Mode" THEN "AI_FQ3205_Bon2_HMI" := 0.0; END_IF;
END_REGION

REGION Network 64: Reset AI_LT3209_Bon2_HMI về 0.0 khi ở chế độ chạy thật
   RUNG wire#powerrail
      I_Contact( "AI_HMI_Sim_Mode" )
      { S7_GenerateENO := "TRUE" } Move(in := 0.0, out1 => "AI_LT3209_Bon2_HMI")
   END_RUNG
   // the same network as SCL:
   IF NOT "AI_HMI_Sim_Mode" THEN "AI_LT3209_Bon2_HMI" := 0.0; END_IF;
END_REGION

REGION Network 65: Reset AI_TT3208_Bon2_HMI về 0.0 khi ở chế độ chạy thật
   RUNG wire#powerrail
      I_Contact( "AI_HMI_Sim_Mode" )
      { S7_GenerateENO := "TRUE" } Move(in := 0.0, out1 => "AI_TT3208_Bon2_HMI")
   END_RUNG
   // the same network as SCL:
   IF NOT "AI_HMI_Sim_Mode" THEN "AI_TT3208_Bon2_HMI" := 0.0; END_IF;
END_REGION

REGION Network 66: Reset AI_LT3302_BonChua1_HMI về 0.0 khi ở chế độ chạy thật
   RUNG wire#powerrail
      I_Contact( "AI_HMI_Sim_Mode" )
      { S7_GenerateENO := "TRUE" } Move(in := 0.0, out1 => "AI_LT3302_BonChua1_HMI")
   END_RUNG
   // the same network as SCL:
   IF NOT "AI_HMI_Sim_Mode" THEN "AI_LT3302_BonChua1_HMI" := 0.0; END_IF;
END_REGION

REGION Network 67: Reset AI_TT3301_BonChua1_HMI về 0.0 khi ở chế độ chạy thật
   RUNG wire#powerrail
      I_Contact( "AI_HMI_Sim_Mode" )
      { S7_GenerateENO := "TRUE" } Move(in := 0.0, out1 => "AI_TT3301_BonChua1_HMI")
   END_RUNG
   // the same network as SCL:
   IF NOT "AI_HMI_Sim_Mode" THEN "AI_TT3301_BonChua1_HMI" := 0.0; END_IF;
END_REGION

REGION Network 68: Reset AI_TT3303_TraoDoiNhiet_HMI về 0.0 khi ở chế độ chạy thật
   RUNG wire#powerrail
      I_Contact( "AI_HMI_Sim_Mode" )
      { S7_GenerateENO := "TRUE" } Move(in := 0.0, out1 => "AI_TT3303_TraoDoiNhiet_HMI")
   END_RUNG
   // the same network as SCL:
   IF NOT "AI_HMI_Sim_Mode" THEN "AI_TT3303_TraoDoiNhiet_HMI" := 0.0; END_IF;
END_REGION

REGION Network 69: Reset AI_LT3307_BonChua2_HMI về 0.0 khi ở chế độ chạy thật
   RUNG wire#powerrail
      I_Contact( "AI_HMI_Sim_Mode" )
      { S7_GenerateENO := "TRUE" } Move(in := 0.0, out1 => "AI_LT3307_BonChua2_HMI")
   END_RUNG
   // the same network as SCL:
   IF NOT "AI_HMI_Sim_Mode" THEN "AI_LT3307_BonChua2_HMI" := 0.0; END_IF;
END_REGION

REGION Network 70: Reset AI_TT3306_BonChua2_HMI về 0.0 khi ở chế độ chạy thật
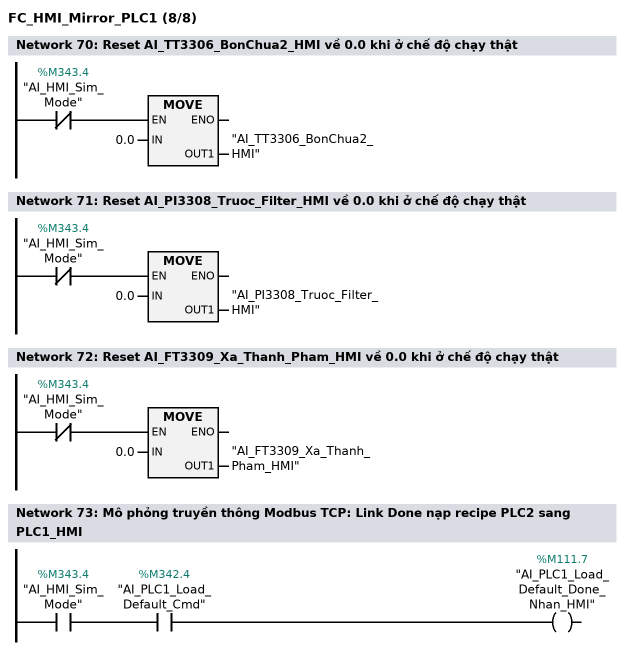
   RUNG wire#powerrail
      I_Contact( "AI_HMI_Sim_Mode" )
      { S7_GenerateENO := "TRUE" } Move(in := 0.0, out1 => "AI_TT3306_BonChua2_HMI")
   END_RUNG
   // the same network as SCL:
   IF NOT "AI_HMI_Sim_Mode" THEN "AI_TT3306_BonChua2_HMI" := 0.0; END_IF;
END_REGION

REGION Network 71: Reset AI_PI3308_Truoc_Filter_HMI về 0.0 khi ở chế độ chạy thật
   RUNG wire#powerrail
      I_Contact( "AI_HMI_Sim_Mode" )
      { S7_GenerateENO := "TRUE" } Move(in := 0.0, out1 => "AI_PI3308_Truoc_Filter_HMI")
   END_RUNG
   // the same network as SCL:
   IF NOT "AI_HMI_Sim_Mode" THEN "AI_PI3308_Truoc_Filter_HMI" := 0.0; END_IF;
END_REGION

REGION Network 72: Reset AI_FT3309_Xa_Thanh_Pham_HMI về 0.0 khi ở chế độ chạy thật
   RUNG wire#powerrail
      I_Contact( "AI_HMI_Sim_Mode" )
      { S7_GenerateENO := "TRUE" } Move(in := 0.0, out1 => "AI_FT3309_Xa_Thanh_Pham_HMI")
   END_RUNG
   // the same network as SCL:
   IF NOT "AI_HMI_Sim_Mode" THEN "AI_FT3309_Xa_Thanh_Pham_HMI" := 0.0; END_IF;
END_REGION

REGION Network 73: Mô phỏng truyền thông Modbus TCP: Link Done nạp recipe PLC2 sang PLC1_HMI
   RUNG wire#powerrail
      Contact( "AI_HMI_Sim_Mode" )
      Contact( "AI_PLC1_Load_Default_Cmd" )
      Coil( "AI_PLC1_Load_Default_Done_Nhan_HMI" )
   END_RUNG
   // the same network as SCL:
   "AI_PLC1_Load_Default_Done_Nhan_HMI" := "AI_HMI_Sim_Mode" AND "AI_PLC1_Load_Default_Cmd";
END_REGION
END_FUNCTION

ORGANIZATION_BLOCK "OB30_PID_PLC1_Bon2"   // OB30, LAD, CyclicInterrupt
{ S7_Optimized_Access := 'TRUE' }
VERSION : 0.1
// stored: AutoNumber true, IsIECCheckEnabled false
   VAR_INPUT
      Initial_Call : Bool;
      Remanence : Bool;
   END_VAR
BEGIN

REGION Network 1: Initialize PID Bon 2 Kp parameter
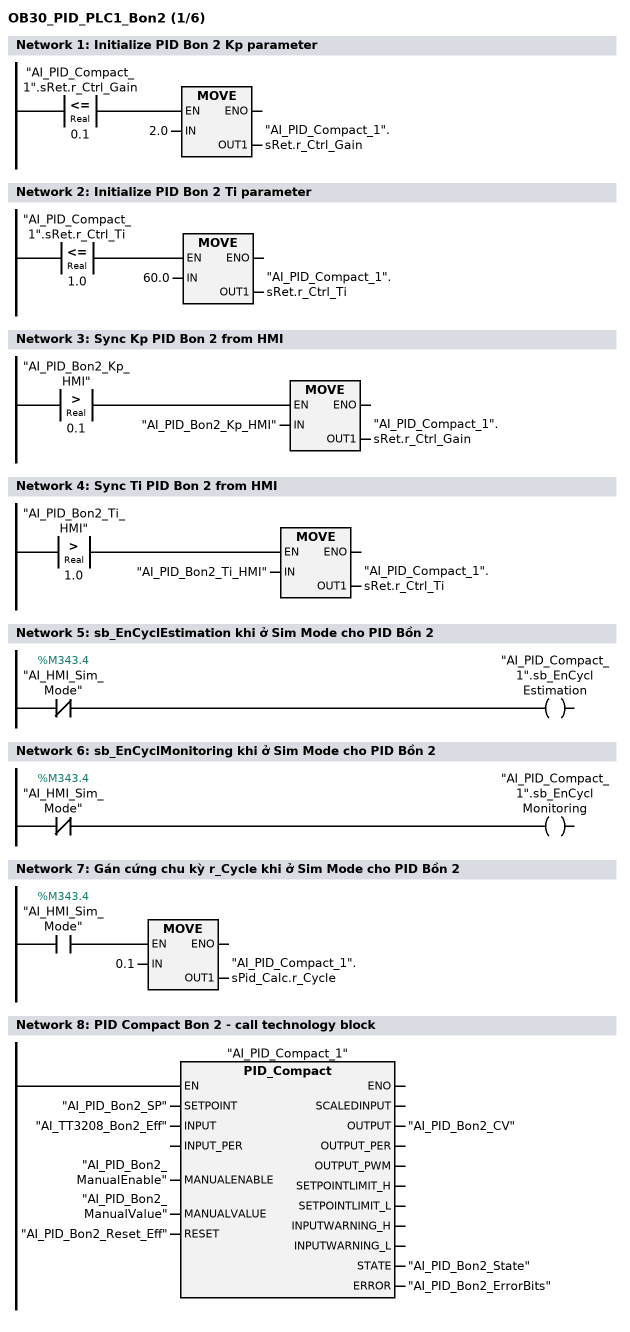
   RUNG wire#powerrail
      { S7_Templates := "SrcType := Real" } LE_Contact(in1 := "AI_PID_Compact_1".sRet.r_Ctrl_Gain, in2 := 0.1)
      { S7_GenerateENO := "TRUE" } Move(in := 2.0, out1 => "AI_PID_Compact_1".sRet.r_Ctrl_Gain)
   END_RUNG
   // the same network as SCL:
   IF "AI_PID_Compact_1".sRet.r_Ctrl_Gain <= 0.1 THEN "AI_PID_Compact_1".sRet.r_Ctrl_Gain := 2.0; END_IF;
END_REGION

REGION Network 2: Initialize PID Bon 2 Ti parameter
   RUNG wire#powerrail
      { S7_Templates := "SrcType := Real" } LE_Contact(in1 := "AI_PID_Compact_1".sRet.r_Ctrl_Ti, in2 := 1.0)
      { S7_GenerateENO := "TRUE" } Move(in := 60.0, out1 => "AI_PID_Compact_1".sRet.r_Ctrl_Ti)
   END_RUNG
   // the same network as SCL:
   IF "AI_PID_Compact_1".sRet.r_Ctrl_Ti <= 1.0 THEN "AI_PID_Compact_1".sRet.r_Ctrl_Ti := 60.0; END_IF;
END_REGION

REGION Network 3: Sync Kp PID Bon 2 from HMI
   RUNG wire#powerrail
      { S7_Templates := "SrcType := Real" } GT_Contact(in1 := "AI_PID_Bon2_Kp_HMI", in2 := 0.1)
      { S7_GenerateENO := "TRUE" } Move(in := "AI_PID_Bon2_Kp_HMI", out1 => "AI_PID_Compact_1".sRet.r_Ctrl_Gain)
   END_RUNG
   // the same network as SCL:
   IF "AI_PID_Bon2_Kp_HMI" > 0.1 THEN "AI_PID_Compact_1".sRet.r_Ctrl_Gain := "AI_PID_Bon2_Kp_HMI"; END_IF;
END_REGION

REGION Network 4: Sync Ti PID Bon 2 from HMI
   RUNG wire#powerrail
      { S7_Templates := "SrcType := Real" } GT_Contact(in1 := "AI_PID_Bon2_Ti_HMI", in2 := 1.0)
      { S7_GenerateENO := "TRUE" } Move(in := "AI_PID_Bon2_Ti_HMI", out1 => "AI_PID_Compact_1".sRet.r_Ctrl_Ti)
   END_RUNG
   // the same network as SCL:
   IF "AI_PID_Bon2_Ti_HMI" > 1.0 THEN "AI_PID_Compact_1".sRet.r_Ctrl_Ti := "AI_PID_Bon2_Ti_HMI"; END_IF;
END_REGION

REGION Network 5: sb_EnCyclEstimation khi ở Sim Mode cho PID Bồn 2
   RUNG wire#powerrail
      I_Contact( "AI_HMI_Sim_Mode" )
      Coil( "AI_PID_Compact_1".sb_EnCyclEstimation )
   END_RUNG
   // the same network as SCL:
   "AI_PID_Compact_1".sb_EnCyclEstimation := NOT "AI_HMI_Sim_Mode";
END_REGION

REGION Network 6: sb_EnCyclMonitoring khi ở Sim Mode cho PID Bồn 2
   RUNG wire#powerrail
      I_Contact( "AI_HMI_Sim_Mode" )
      Coil( "AI_PID_Compact_1".sb_EnCyclMonitoring )
   END_RUNG
   // the same network as SCL:
   "AI_PID_Compact_1".sb_EnCyclMonitoring := NOT "AI_HMI_Sim_Mode";
END_REGION

REGION Network 7: Gán cứng chu kỳ r_Cycle khi ở Sim Mode cho PID Bồn 2
   RUNG wire#powerrail
      Contact( "AI_HMI_Sim_Mode" )
      { S7_GenerateENO := "TRUE" } Move(in := 0.1, out1 => "AI_PID_Compact_1".sPid_Calc.r_Cycle)
   END_RUNG
   // the same network as SCL:
   IF "AI_HMI_Sim_Mode" THEN "AI_PID_Compact_1".sPid_Calc.r_Cycle := 0.1; END_IF;
END_REGION

REGION Network 8: PID Compact Bon 2 - call technology block
   RUNG wire#powerrail
      "AI_PID_Compact_1".PID_Compact(Setpoint := "AI_PID_Bon2_SP", Input := "AI_TT3208_Bon2_Eff", Input_PER :=, ManualEnable := "AI_PID_Bon2_ManualEnable", ManualValue := "AI_PID_Bon2_ManualValue", Reset := "AI_PID_Bon2_Reset_Eff", ScaledInput =>, Output => "AI_PID_Bon2_CV", Output_PER =>, Output_PWM =>, SetpointLimit_H =>, SetpointLimit_L =>, InputWarning_H =>, InputWarning_L =>, State => "AI_PID_Bon2_State", Error => "AI_PID_Bon2_ErrorBits")
   END_RUNG
   // the same network as SCL:
   "AI_PID_Compact_1"(Setpoint := "AI_PID_Bon2_SP",   // PID_Compact
                      Input := "AI_TT3208_Bon2_Eff",
                      ManualEnable := "AI_PID_Bon2_ManualEnable",
                      ManualValue := "AI_PID_Bon2_ManualValue",
                      Reset := "AI_PID_Bon2_Reset_Eff",
                      Output => "AI_PID_Bon2_CV",
                      State => "AI_PID_Bon2_State",
                      Error => "AI_PID_Bon2_ErrorBits");
END_REGION

REGION Network 9: Detect PID Bon 2 Error
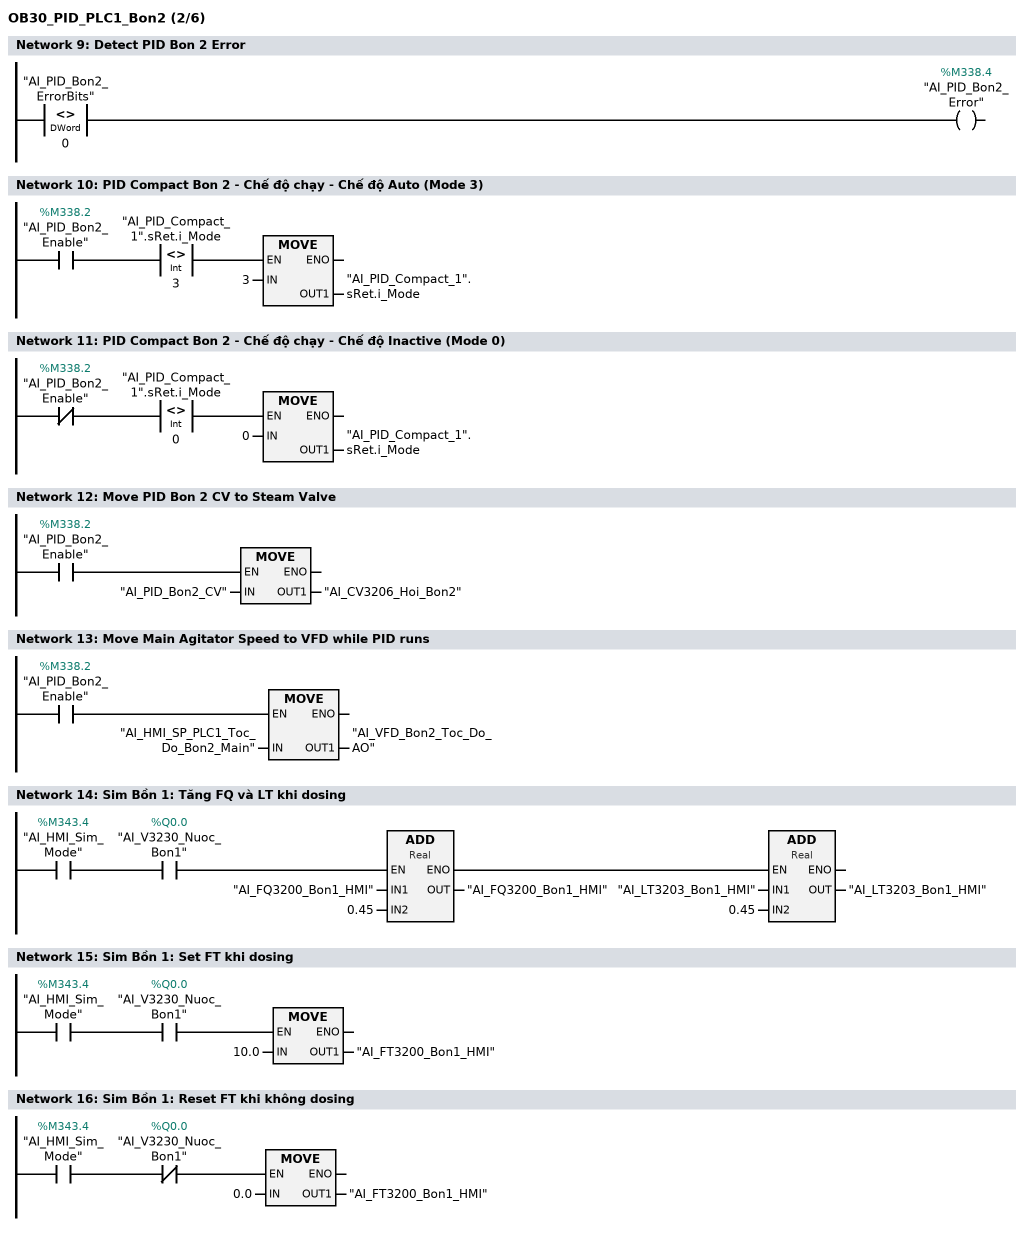
   RUNG wire#powerrail
      { S7_Templates := "SrcType := DWord" } NE_Contact(in1 := "AI_PID_Bon2_ErrorBits", in2 := 0)
      Coil( "AI_PID_Bon2_Error" )
   END_RUNG
   // the same network as SCL:
   "AI_PID_Bon2_Error" := "AI_PID_Bon2_ErrorBits" <> 0;
END_REGION

REGION Network 10: PID Compact Bon 2 - Chế độ chạy - Chế độ Auto (Mode 3)
   RUNG wire#powerrail
      Contact( "AI_PID_Bon2_Enable" )
      { S7_Templates := "SrcType := Int" } NE_Contact(in1 := "AI_PID_Compact_1".sRet.i_Mode, in2 := 3)
      { S7_GenerateENO := "TRUE" } Move(in := 3, out1 => "AI_PID_Compact_1".sRet.i_Mode)
   END_RUNG
   // the same network as SCL:
   IF "AI_PID_Bon2_Enable" AND ("AI_PID_Compact_1".sRet.i_Mode <> 3) THEN
       "AI_PID_Compact_1".sRet.i_Mode := 3;
   END_IF;
END_REGION

REGION Network 11: PID Compact Bon 2 - Chế độ chạy - Chế độ Inactive (Mode 0)
   RUNG wire#powerrail
      I_Contact( "AI_PID_Bon2_Enable" )
      { S7_Templates := "SrcType := Int" } NE_Contact(in1 := "AI_PID_Compact_1".sRet.i_Mode, in2 := 0)
      { S7_GenerateENO := "TRUE" } Move(in := 0, out1 => "AI_PID_Compact_1".sRet.i_Mode)
   END_RUNG
   // the same network as SCL:
   IF NOT "AI_PID_Bon2_Enable" AND ("AI_PID_Compact_1".sRet.i_Mode <> 0) THEN
       "AI_PID_Compact_1".sRet.i_Mode := 0;
   END_IF;
END_REGION

REGION Network 12: Move PID Bon 2 CV to Steam Valve
   RUNG wire#powerrail
      Contact( "AI_PID_Bon2_Enable" )
      { S7_GenerateENO := "TRUE" } Move(in := "AI_PID_Bon2_CV", out1 => "AI_CV3206_Hoi_Bon2")
   END_RUNG
   // the same network as SCL:
   IF "AI_PID_Bon2_Enable" THEN "AI_CV3206_Hoi_Bon2" := "AI_PID_Bon2_CV"; END_IF;
END_REGION

REGION Network 13: Move Main Agitator Speed to VFD while PID runs
   RUNG wire#powerrail
      Contact( "AI_PID_Bon2_Enable" )
      { S7_GenerateENO := "TRUE" } Move(in := "AI_HMI_SP_PLC1_Toc_Do_Bon2_Main", out1 => "AI_VFD_Bon2_Toc_Do_AO")
   END_RUNG
   // the same network as SCL:
   IF "AI_PID_Bon2_Enable" THEN "AI_VFD_Bon2_Toc_Do_AO" := "AI_HMI_SP_PLC1_Toc_Do_Bon2_Main"; END_IF;
END_REGION

REGION Network 14: Sim Bồn 1: Tăng FQ và LT khi dosing
   RUNG wire#powerrail
      Contact( "AI_HMI_Sim_Mode" )
      Contact( "AI_V3230_Nuoc_Bon1" )
      { S7_Templates := "SrcType := Real"; S7_GenerateENO := "TRUE" } Add(in1 := "AI_FQ3200_Bon1_HMI", in2 := 0.45, out => "AI_FQ3200_Bon1_HMI")
      { S7_Templates := "SrcType := Real"; S7_GenerateENO := "TRUE" } Add(in1 := "AI_LT3203_Bon1_HMI", in2 := 0.45, out => "AI_LT3203_Bon1_HMI")
   END_RUNG
   // the same network as SCL:
   // ENO of a box is taken as its EN; it also drops when the box reports an error
   IF "AI_HMI_Sim_Mode" AND "AI_V3230_Nuoc_Bon1" THEN
       "AI_FQ3200_Bon1_HMI" := "AI_FQ3200_Bon1_HMI" + 0.45;
       "AI_LT3203_Bon1_HMI" := "AI_LT3203_Bon1_HMI" + 0.45;
   END_IF;
END_REGION

REGION Network 15: Sim Bồn 1: Set FT khi dosing
   RUNG wire#powerrail
      Contact( "AI_HMI_Sim_Mode" )
      Contact( "AI_V3230_Nuoc_Bon1" )
      { S7_GenerateENO := "TRUE" } Move(in := 10.0, out1 => "AI_FT3200_Bon1_HMI")
   END_RUNG
   // the same network as SCL:
   IF "AI_HMI_Sim_Mode" AND "AI_V3230_Nuoc_Bon1" THEN "AI_FT3200_Bon1_HMI" := 10.0; END_IF;
END_REGION

REGION Network 16: Sim Bồn 1: Reset FT khi không dosing
   RUNG wire#powerrail
      Contact( "AI_HMI_Sim_Mode" )
      I_Contact( "AI_V3230_Nuoc_Bon1" )
      { S7_GenerateENO := "TRUE" } Move(in := 0.0, out1 => "AI_FT3200_Bon1_HMI")
   END_RUNG
   // the same network as SCL:
   IF "AI_HMI_Sim_Mode" AND NOT "AI_V3230_Nuoc_Bon1" THEN "AI_FT3200_Bon1_HMI" := 0.0; END_IF;
END_REGION

REGION Network 17: Sim Bồn 1: Giảm LT khi xả đáy
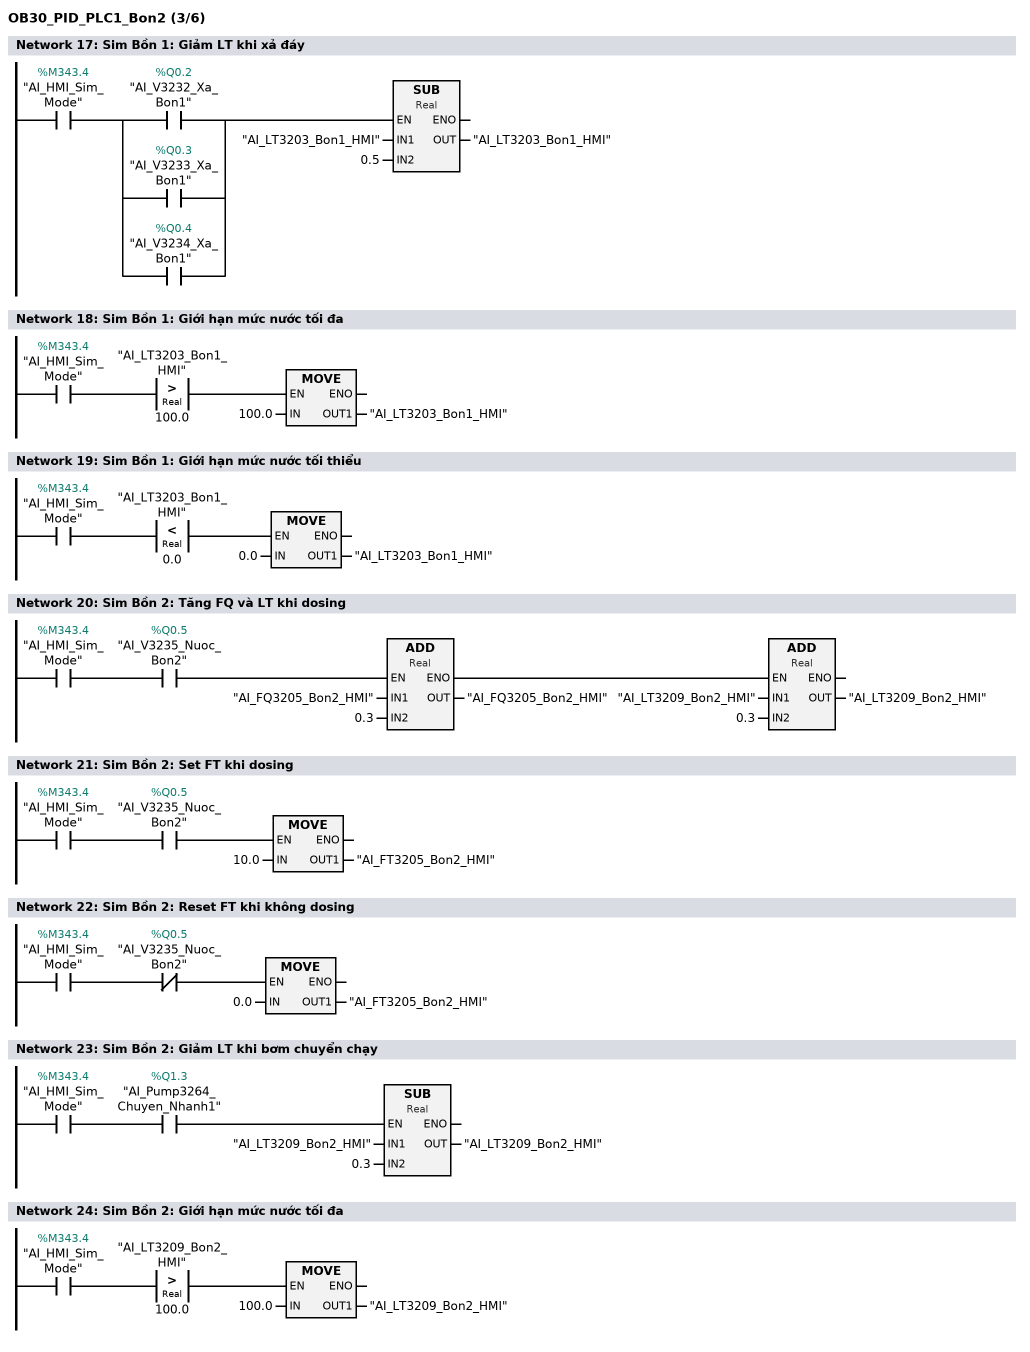
   RUNG wire#powerrail
      Contact( "AI_HMI_Sim_Mode" )
      wire#w1
      Contact( "AI_V3232_Xa_Bon1" )
      wire#w2
      { S7_Templates := "SrcType := Real"; S7_GenerateENO := "TRUE" } Sub(in1 := "AI_LT3203_Bon1_HMI", in2 := 0.5, out => "AI_LT3203_Bon1_HMI")
   END_RUNG
   RUNG wire#w1
      Contact( "AI_V3233_Xa_Bon1" )
   END_RUNG wire#w2
   RUNG wire#w1
      Contact( "AI_V3234_Xa_Bon1" )
   END_RUNG wire#w2
   // the same network as SCL:
   IF "AI_HMI_Sim_Mode" AND ("AI_V3232_Xa_Bon1" OR "AI_V3233_Xa_Bon1" OR "AI_V3234_Xa_Bon1") THEN
       "AI_LT3203_Bon1_HMI" := "AI_LT3203_Bon1_HMI" - 0.5;
   END_IF;
END_REGION

REGION Network 18: Sim Bồn 1: Giới hạn mức nước tối đa
   RUNG wire#powerrail
      Contact( "AI_HMI_Sim_Mode" )
      { S7_Templates := "SrcType := Real" } GT_Contact(in1 := "AI_LT3203_Bon1_HMI", in2 := 100.0)
      { S7_GenerateENO := "TRUE" } Move(in := 100.0, out1 => "AI_LT3203_Bon1_HMI")
   END_RUNG
   // the same network as SCL:
   IF "AI_HMI_Sim_Mode" AND ("AI_LT3203_Bon1_HMI" > 100.0) THEN "AI_LT3203_Bon1_HMI" := 100.0; END_IF;
END_REGION

REGION Network 19: Sim Bồn 1: Giới hạn mức nước tối thiểu
   RUNG wire#powerrail
      Contact( "AI_HMI_Sim_Mode" )
      { S7_Templates := "SrcType := Real" } LT_Contact(in1 := "AI_LT3203_Bon1_HMI", in2 := 0.0)
      { S7_GenerateENO := "TRUE" } Move(in := 0.0, out1 => "AI_LT3203_Bon1_HMI")
   END_RUNG
   // the same network as SCL:
   IF "AI_HMI_Sim_Mode" AND ("AI_LT3203_Bon1_HMI" < 0.0) THEN "AI_LT3203_Bon1_HMI" := 0.0; END_IF;
END_REGION

REGION Network 20: Sim Bồn 2: Tăng FQ và LT khi dosing
   RUNG wire#powerrail
      Contact( "AI_HMI_Sim_Mode" )
      Contact( "AI_V3235_Nuoc_Bon2" )
      { S7_Templates := "SrcType := Real"; S7_GenerateENO := "TRUE" } Add(in1 := "AI_FQ3205_Bon2_HMI", in2 := 0.3, out => "AI_FQ3205_Bon2_HMI")
      { S7_Templates := "SrcType := Real"; S7_GenerateENO := "TRUE" } Add(in1 := "AI_LT3209_Bon2_HMI", in2 := 0.3, out => "AI_LT3209_Bon2_HMI")
   END_RUNG
   // the same network as SCL:
   // ENO of a box is taken as its EN; it also drops when the box reports an error
   IF "AI_HMI_Sim_Mode" AND "AI_V3235_Nuoc_Bon2" THEN
       "AI_FQ3205_Bon2_HMI" := "AI_FQ3205_Bon2_HMI" + 0.3;
       "AI_LT3209_Bon2_HMI" := "AI_LT3209_Bon2_HMI" + 0.3;
   END_IF;
END_REGION

REGION Network 21: Sim Bồn 2: Set FT khi dosing
   RUNG wire#powerrail
      Contact( "AI_HMI_Sim_Mode" )
      Contact( "AI_V3235_Nuoc_Bon2" )
      { S7_GenerateENO := "TRUE" } Move(in := 10.0, out1 => "AI_FT3205_Bon2_HMI")
   END_RUNG
   // the same network as SCL:
   IF "AI_HMI_Sim_Mode" AND "AI_V3235_Nuoc_Bon2" THEN "AI_FT3205_Bon2_HMI" := 10.0; END_IF;
END_REGION

REGION Network 22: Sim Bồn 2: Reset FT khi không dosing
   RUNG wire#powerrail
      Contact( "AI_HMI_Sim_Mode" )
      I_Contact( "AI_V3235_Nuoc_Bon2" )
      { S7_GenerateENO := "TRUE" } Move(in := 0.0, out1 => "AI_FT3205_Bon2_HMI")
   END_RUNG
   // the same network as SCL:
   IF "AI_HMI_Sim_Mode" AND NOT "AI_V3235_Nuoc_Bon2" THEN "AI_FT3205_Bon2_HMI" := 0.0; END_IF;
END_REGION

REGION Network 23: Sim Bồn 2: Giảm LT khi bơm chuyển chạy
   RUNG wire#powerrail
      Contact( "AI_HMI_Sim_Mode" )
      Contact( "AI_Pump3264_Chuyen_Nhanh1" )
      { S7_Templates := "SrcType := Real"; S7_GenerateENO := "TRUE" } Sub(in1 := "AI_LT3209_Bon2_HMI", in2 := 0.3, out => "AI_LT3209_Bon2_HMI")
   END_RUNG
   // the same network as SCL:
   IF "AI_HMI_Sim_Mode" AND "AI_Pump3264_Chuyen_Nhanh1" THEN
       "AI_LT3209_Bon2_HMI" := "AI_LT3209_Bon2_HMI" - 0.3;
   END_IF;
END_REGION

REGION Network 24: Sim Bồn 2: Giới hạn mức nước tối đa
   RUNG wire#powerrail
      Contact( "AI_HMI_Sim_Mode" )
      { S7_Templates := "SrcType := Real" } GT_Contact(in1 := "AI_LT3209_Bon2_HMI", in2 := 100.0)
      { S7_GenerateENO := "TRUE" } Move(in := 100.0, out1 => "AI_LT3209_Bon2_HMI")
   END_RUNG
   // the same network as SCL:
   IF "AI_HMI_Sim_Mode" AND ("AI_LT3209_Bon2_HMI" > 100.0) THEN "AI_LT3209_Bon2_HMI" := 100.0; END_IF;
END_REGION

REGION Network 25: Sim Bồn 2: Giới hạn mức nước tối thiểu
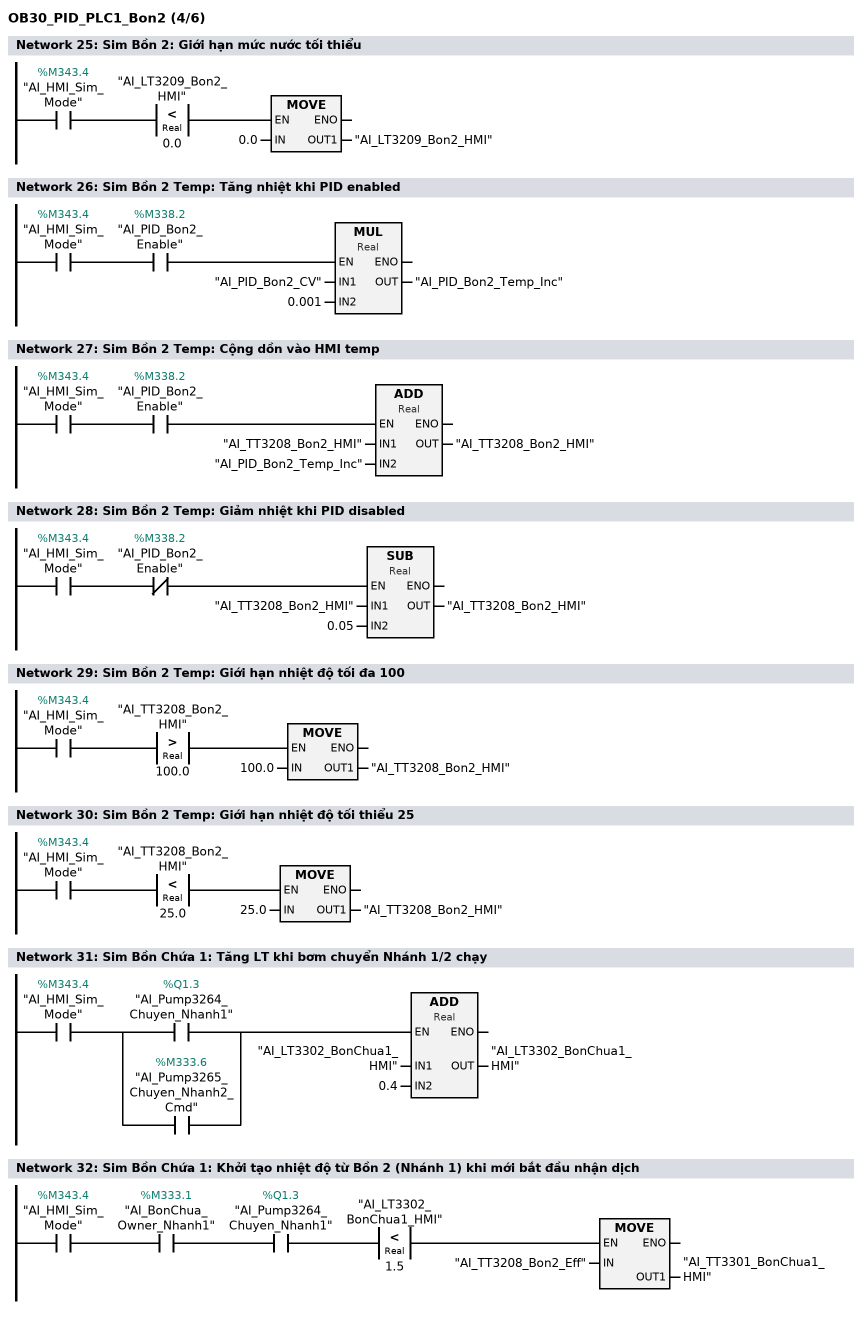
   RUNG wire#powerrail
      Contact( "AI_HMI_Sim_Mode" )
      { S7_Templates := "SrcType := Real" } LT_Contact(in1 := "AI_LT3209_Bon2_HMI", in2 := 0.0)
      { S7_GenerateENO := "TRUE" } Move(in := 0.0, out1 => "AI_LT3209_Bon2_HMI")
   END_RUNG
   // the same network as SCL:
   IF "AI_HMI_Sim_Mode" AND ("AI_LT3209_Bon2_HMI" < 0.0) THEN "AI_LT3209_Bon2_HMI" := 0.0; END_IF;
END_REGION

REGION Network 26: Sim Bồn 2 Temp: Tăng nhiệt khi PID enabled
   RUNG wire#powerrail
      Contact( "AI_HMI_Sim_Mode" )
      Contact( "AI_PID_Bon2_Enable" )
      { S7_Templates := "SrcType := Real"; S7_GenerateENO := "TRUE" } Mul(in1 := "AI_PID_Bon2_CV", in2 := 0.001, out => "AI_PID_Bon2_Temp_Inc")
   END_RUNG
   // the same network as SCL:
   IF "AI_HMI_Sim_Mode" AND "AI_PID_Bon2_Enable" THEN
       "AI_PID_Bon2_Temp_Inc" := "AI_PID_Bon2_CV" * 0.001;
   END_IF;
END_REGION

REGION Network 27: Sim Bồn 2 Temp: Cộng dồn vào HMI temp
   RUNG wire#powerrail
      Contact( "AI_HMI_Sim_Mode" )
      Contact( "AI_PID_Bon2_Enable" )
      { S7_Templates := "SrcType := Real"; S7_GenerateENO := "TRUE" } Add(in1 := "AI_TT3208_Bon2_HMI", in2 := "AI_PID_Bon2_Temp_Inc", out => "AI_TT3208_Bon2_HMI")
   END_RUNG
   // the same network as SCL:
   IF "AI_HMI_Sim_Mode" AND "AI_PID_Bon2_Enable" THEN
       "AI_TT3208_Bon2_HMI" := "AI_TT3208_Bon2_HMI" + "AI_PID_Bon2_Temp_Inc";
   END_IF;
END_REGION

REGION Network 28: Sim Bồn 2 Temp: Giảm nhiệt khi PID disabled
   RUNG wire#powerrail
      Contact( "AI_HMI_Sim_Mode" )
      I_Contact( "AI_PID_Bon2_Enable" )
      { S7_Templates := "SrcType := Real"; S7_GenerateENO := "TRUE" } Sub(in1 := "AI_TT3208_Bon2_HMI", in2 := 0.05, out => "AI_TT3208_Bon2_HMI")
   END_RUNG
   // the same network as SCL:
   IF "AI_HMI_Sim_Mode" AND NOT "AI_PID_Bon2_Enable" THEN
       "AI_TT3208_Bon2_HMI" := "AI_TT3208_Bon2_HMI" - 0.05;
   END_IF;
END_REGION

REGION Network 29: Sim Bồn 2 Temp: Giới hạn nhiệt độ tối đa 100
   RUNG wire#powerrail
      Contact( "AI_HMI_Sim_Mode" )
      { S7_Templates := "SrcType := Real" } GT_Contact(in1 := "AI_TT3208_Bon2_HMI", in2 := 100.0)
      { S7_GenerateENO := "TRUE" } Move(in := 100.0, out1 => "AI_TT3208_Bon2_HMI")
   END_RUNG
   // the same network as SCL:
   IF "AI_HMI_Sim_Mode" AND ("AI_TT3208_Bon2_HMI" > 100.0) THEN "AI_TT3208_Bon2_HMI" := 100.0; END_IF;
END_REGION

REGION Network 30: Sim Bồn 2 Temp: Giới hạn nhiệt độ tối thiểu 25
   RUNG wire#powerrail
      Contact( "AI_HMI_Sim_Mode" )
      { S7_Templates := "SrcType := Real" } LT_Contact(in1 := "AI_TT3208_Bon2_HMI", in2 := 25.0)
      { S7_GenerateENO := "TRUE" } Move(in := 25.0, out1 => "AI_TT3208_Bon2_HMI")
   END_RUNG
   // the same network as SCL:
   IF "AI_HMI_Sim_Mode" AND ("AI_TT3208_Bon2_HMI" < 25.0) THEN "AI_TT3208_Bon2_HMI" := 25.0; END_IF;
END_REGION

REGION Network 31: Sim Bồn Chứa 1: Tăng LT khi bơm chuyển Nhánh 1/2 chạy
   RUNG wire#powerrail
      Contact( "AI_HMI_Sim_Mode" )
      wire#w1
      Contact( "AI_Pump3264_Chuyen_Nhanh1" )
      wire#w2
      { S7_Templates := "SrcType := Real"; S7_GenerateENO := "TRUE" } Add(in1 := "AI_LT3302_BonChua1_HMI", in2 := 0.4, out => "AI_LT3302_BonChua1_HMI")
   END_RUNG
   RUNG wire#w1
      Contact( "AI_Pump3265_Chuyen_Nhanh2_Cmd" )
   END_RUNG wire#w2
   // the same network as SCL:
   IF "AI_HMI_Sim_Mode" AND ("AI_Pump3264_Chuyen_Nhanh1" OR "AI_Pump3265_Chuyen_Nhanh2_Cmd") THEN
       "AI_LT3302_BonChua1_HMI" := "AI_LT3302_BonChua1_HMI" + 0.4;
   END_IF;
END_REGION

REGION Network 32: Sim Bồn Chứa 1: Khởi tạo nhiệt độ từ Bồn 2 (Nhánh 1) khi mới bắt đầu nhận dịch
   RUNG wire#powerrail
      Contact( "AI_HMI_Sim_Mode" )
      Contact( "AI_BonChua_Owner_Nhanh1" )
      Contact( "AI_Pump3264_Chuyen_Nhanh1" )
      { S7_Templates := "SrcType := Real" } LT_Contact(in1 := "AI_LT3302_BonChua1_HMI", in2 := 1.5)
      { S7_GenerateENO := "TRUE" } Move(in := "AI_TT3208_Bon2_Eff", out1 => "AI_TT3301_BonChua1_HMI")
   END_RUNG
   // the same network as SCL:
   IF "AI_HMI_Sim_Mode" AND "AI_BonChua_Owner_Nhanh1" AND "AI_Pump3264_Chuyen_Nhanh1" AND ("AI_LT3302_BonChua1_HMI" < 1.5) THEN
       "AI_TT3301_BonChua1_HMI" := "AI_TT3208_Bon2_Eff";
   END_IF;
END_REGION

REGION Network 33: Sim Bồn Chứa 1: Khởi tạo nhiệt độ từ Bồn 4 (Nhánh 2) khi mới bắt đầu nhận dịch
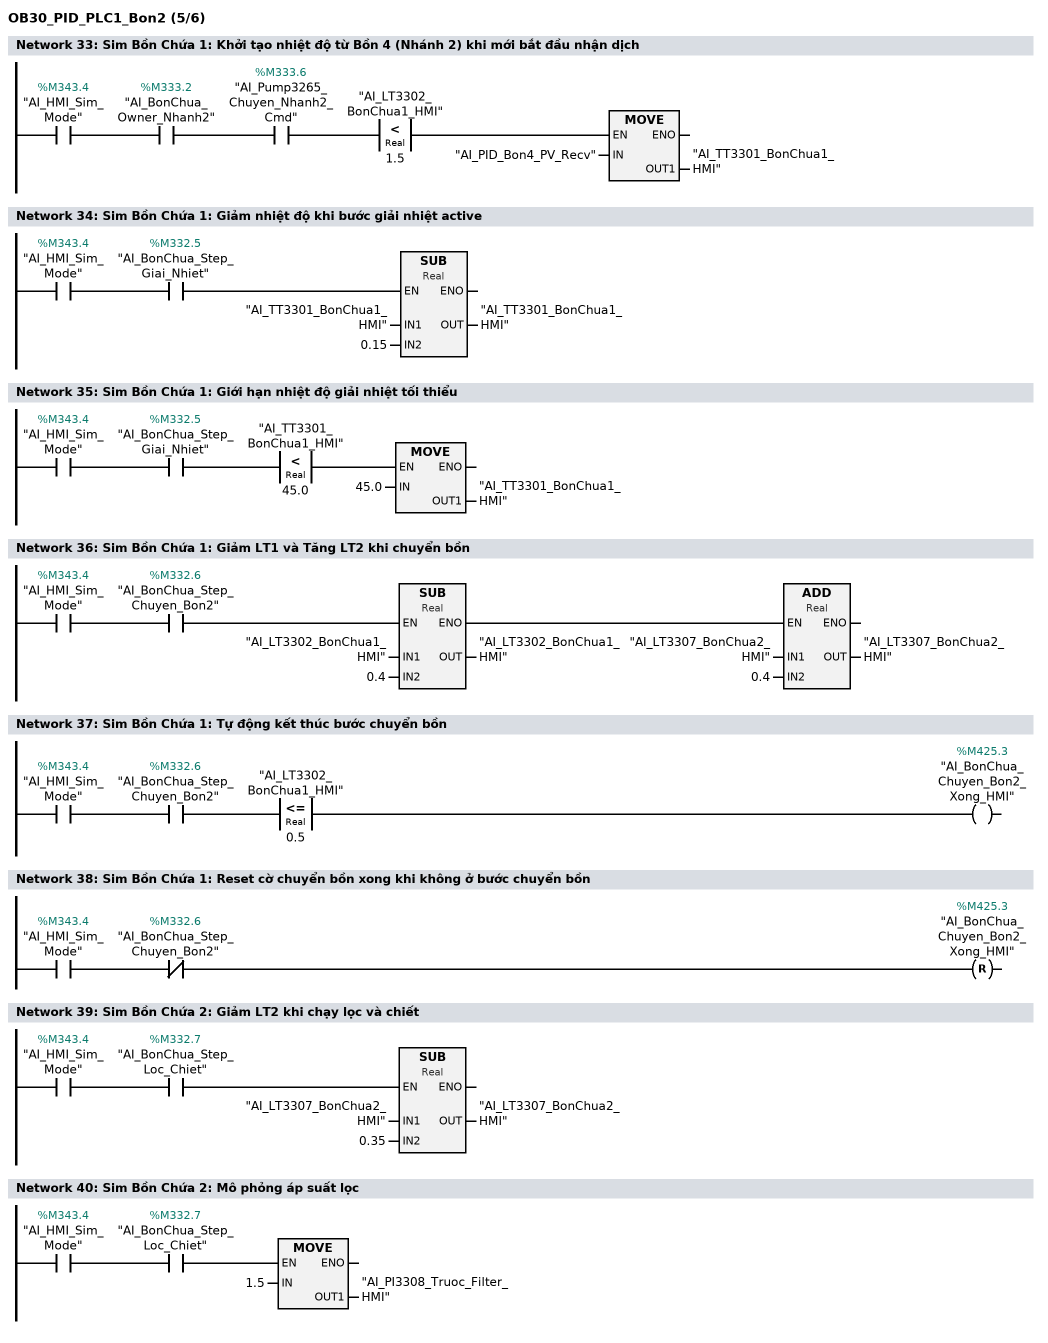
   RUNG wire#powerrail
      Contact( "AI_HMI_Sim_Mode" )
      Contact( "AI_BonChua_Owner_Nhanh2" )
      Contact( "AI_Pump3265_Chuyen_Nhanh2_Cmd" )
      { S7_Templates := "SrcType := Real" } LT_Contact(in1 := "AI_LT3302_BonChua1_HMI", in2 := 1.5)
      { S7_GenerateENO := "TRUE" } Move(in := "AI_PID_Bon4_PV_Recv", out1 => "AI_TT3301_BonChua1_HMI")
   END_RUNG
   // the same network as SCL:
   IF "AI_HMI_Sim_Mode" AND "AI_BonChua_Owner_Nhanh2" AND "AI_Pump3265_Chuyen_Nhanh2_Cmd" AND ("AI_LT3302_BonChua1_HMI" < 1.5) THEN
       "AI_TT3301_BonChua1_HMI" := "AI_PID_Bon4_PV_Recv";
   END_IF;
END_REGION

REGION Network 34: Sim Bồn Chứa 1: Giảm nhiệt độ khi bước giải nhiệt active
   RUNG wire#powerrail
      Contact( "AI_HMI_Sim_Mode" )
      Contact( "AI_BonChua_Step_Giai_Nhiet" )
      { S7_Templates := "SrcType := Real"; S7_GenerateENO := "TRUE" } Sub(in1 := "AI_TT3301_BonChua1_HMI", in2 := 0.15, out => "AI_TT3301_BonChua1_HMI")
   END_RUNG
   // the same network as SCL:
   IF "AI_HMI_Sim_Mode" AND "AI_BonChua_Step_Giai_Nhiet" THEN
       "AI_TT3301_BonChua1_HMI" := "AI_TT3301_BonChua1_HMI" - 0.15;
   END_IF;
END_REGION

REGION Network 35: Sim Bồn Chứa 1: Giới hạn nhiệt độ giải nhiệt tối thiểu
   RUNG wire#powerrail
      Contact( "AI_HMI_Sim_Mode" )
      Contact( "AI_BonChua_Step_Giai_Nhiet" )
      { S7_Templates := "SrcType := Real" } LT_Contact(in1 := "AI_TT3301_BonChua1_HMI", in2 := 45.0)
      { S7_GenerateENO := "TRUE" } Move(in := 45.0, out1 => "AI_TT3301_BonChua1_HMI")
   END_RUNG
   // the same network as SCL:
   IF "AI_HMI_Sim_Mode" AND "AI_BonChua_Step_Giai_Nhiet" AND ("AI_TT3301_BonChua1_HMI" < 45.0) THEN
       "AI_TT3301_BonChua1_HMI" := 45.0;
   END_IF;
END_REGION

REGION Network 36: Sim Bồn Chứa 1: Giảm LT1 và Tăng LT2 khi chuyển bồn
   RUNG wire#powerrail
      Contact( "AI_HMI_Sim_Mode" )
      Contact( "AI_BonChua_Step_Chuyen_Bon2" )
      { S7_Templates := "SrcType := Real"; S7_GenerateENO := "TRUE" } Sub(in1 := "AI_LT3302_BonChua1_HMI", in2 := 0.4, out => "AI_LT3302_BonChua1_HMI")
      { S7_Templates := "SrcType := Real"; S7_GenerateENO := "TRUE" } Add(in1 := "AI_LT3307_BonChua2_HMI", in2 := 0.4, out => "AI_LT3307_BonChua2_HMI")
   END_RUNG
   // the same network as SCL:
   // ENO of a box is taken as its EN; it also drops when the box reports an error
   IF "AI_HMI_Sim_Mode" AND "AI_BonChua_Step_Chuyen_Bon2" THEN
       "AI_LT3302_BonChua1_HMI" := "AI_LT3302_BonChua1_HMI" - 0.4;
       "AI_LT3307_BonChua2_HMI" := "AI_LT3307_BonChua2_HMI" + 0.4;
   END_IF;
END_REGION

REGION Network 37: Sim Bồn Chứa 1: Tự động kết thúc bước chuyển bồn
   RUNG wire#powerrail
      Contact( "AI_HMI_Sim_Mode" )
      Contact( "AI_BonChua_Step_Chuyen_Bon2" )
      { S7_Templates := "SrcType := Real" } LE_Contact(in1 := "AI_LT3302_BonChua1_HMI", in2 := 0.5)
      Coil( "AI_BonChua_Chuyen_Bon2_Xong_HMI" )
   END_RUNG
   // the same network as SCL:
   "AI_BonChua_Chuyen_Bon2_Xong_HMI" := "AI_HMI_Sim_Mode" AND "AI_BonChua_Step_Chuyen_Bon2" AND ("AI_LT3302_BonChua1_HMI" <= 0.5);
END_REGION

REGION Network 38: Sim Bồn Chứa 1: Reset cờ chuyển bồn xong khi không ở bước chuyển bồn
   RUNG wire#powerrail
      Contact( "AI_HMI_Sim_Mode" )
      I_Contact( "AI_BonChua_Step_Chuyen_Bon2" )
      R_Coil( "AI_BonChua_Chuyen_Bon2_Xong_HMI" )
   END_RUNG
   // the same network as SCL:
   IF "AI_HMI_Sim_Mode" AND NOT "AI_BonChua_Step_Chuyen_Bon2" THEN
       "AI_BonChua_Chuyen_Bon2_Xong_HMI" := FALSE;
   END_IF;
END_REGION

REGION Network 39: Sim Bồn Chứa 2: Giảm LT2 khi chạy lọc và chiết
   RUNG wire#powerrail
      Contact( "AI_HMI_Sim_Mode" )
      Contact( "AI_BonChua_Step_Loc_Chiet" )
      { S7_Templates := "SrcType := Real"; S7_GenerateENO := "TRUE" } Sub(in1 := "AI_LT3307_BonChua2_HMI", in2 := 0.35, out => "AI_LT3307_BonChua2_HMI")
   END_RUNG
   // the same network as SCL:
   IF "AI_HMI_Sim_Mode" AND "AI_BonChua_Step_Loc_Chiet" THEN
       "AI_LT3307_BonChua2_HMI" := "AI_LT3307_BonChua2_HMI" - 0.35;
   END_IF;
END_REGION

REGION Network 40: Sim Bồn Chứa 2: Mô phỏng áp suất lọc
   RUNG wire#powerrail
      Contact( "AI_HMI_Sim_Mode" )
      Contact( "AI_BonChua_Step_Loc_Chiet" )
      { S7_GenerateENO := "TRUE" } Move(in := 1.5, out1 => "AI_PI3308_Truoc_Filter_HMI")
   END_RUNG
   // the same network as SCL:
   IF "AI_HMI_Sim_Mode" AND "AI_BonChua_Step_Loc_Chiet" THEN "AI_PI3308_Truoc_Filter_HMI" := 1.5; END_IF;
END_REGION

REGION Network 41: Sim Bồn Chứa 2: Mô phỏng lưu lượng xả
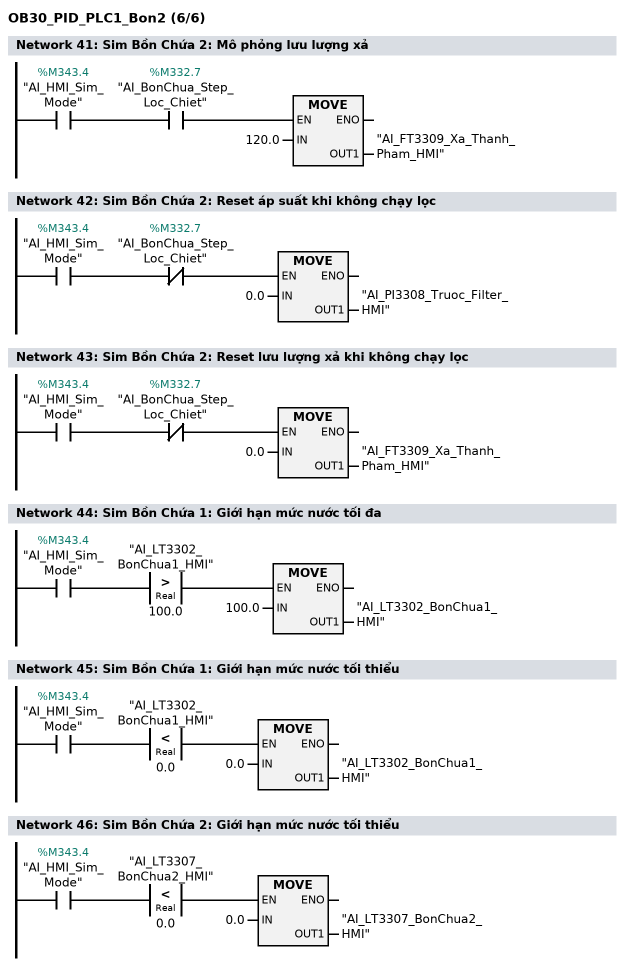
   RUNG wire#powerrail
      Contact( "AI_HMI_Sim_Mode" )
      Contact( "AI_BonChua_Step_Loc_Chiet" )
      { S7_GenerateENO := "TRUE" } Move(in := 120.0, out1 => "AI_FT3309_Xa_Thanh_Pham_HMI")
   END_RUNG
   // the same network as SCL:
   IF "AI_HMI_Sim_Mode" AND "AI_BonChua_Step_Loc_Chiet" THEN "AI_FT3309_Xa_Thanh_Pham_HMI" := 120.0; END_IF;
END_REGION

REGION Network 42: Sim Bồn Chứa 2: Reset áp suất khi không chạy lọc
   RUNG wire#powerrail
      Contact( "AI_HMI_Sim_Mode" )
      I_Contact( "AI_BonChua_Step_Loc_Chiet" )
      { S7_GenerateENO := "TRUE" } Move(in := 0.0, out1 => "AI_PI3308_Truoc_Filter_HMI")
   END_RUNG
   // the same network as SCL:
   IF "AI_HMI_Sim_Mode" AND NOT "AI_BonChua_Step_Loc_Chiet" THEN "AI_PI3308_Truoc_Filter_HMI" := 0.0; END_IF;
END_REGION

REGION Network 43: Sim Bồn Chứa 2: Reset lưu lượng xả khi không chạy lọc
   RUNG wire#powerrail
      Contact( "AI_HMI_Sim_Mode" )
      I_Contact( "AI_BonChua_Step_Loc_Chiet" )
      { S7_GenerateENO := "TRUE" } Move(in := 0.0, out1 => "AI_FT3309_Xa_Thanh_Pham_HMI")
   END_RUNG
   // the same network as SCL:
   IF "AI_HMI_Sim_Mode" AND NOT "AI_BonChua_Step_Loc_Chiet" THEN
       "AI_FT3309_Xa_Thanh_Pham_HMI" := 0.0;
   END_IF;
END_REGION

REGION Network 44: Sim Bồn Chứa 1: Giới hạn mức nước tối đa
   RUNG wire#powerrail
      Contact( "AI_HMI_Sim_Mode" )
      { S7_Templates := "SrcType := Real" } GT_Contact(in1 := "AI_LT3302_BonChua1_HMI", in2 := 100.0)
      { S7_GenerateENO := "TRUE" } Move(in := 100.0, out1 => "AI_LT3302_BonChua1_HMI")
   END_RUNG
   // the same network as SCL:
   IF "AI_HMI_Sim_Mode" AND ("AI_LT3302_BonChua1_HMI" > 100.0) THEN
       "AI_LT3302_BonChua1_HMI" := 100.0;
   END_IF;
END_REGION

REGION Network 45: Sim Bồn Chứa 1: Giới hạn mức nước tối thiểu
   RUNG wire#powerrail
      Contact( "AI_HMI_Sim_Mode" )
      { S7_Templates := "SrcType := Real" } LT_Contact(in1 := "AI_LT3302_BonChua1_HMI", in2 := 0.0)
      { S7_GenerateENO := "TRUE" } Move(in := 0.0, out1 => "AI_LT3302_BonChua1_HMI")
   END_RUNG
   // the same network as SCL:
   IF "AI_HMI_Sim_Mode" AND ("AI_LT3302_BonChua1_HMI" < 0.0) THEN "AI_LT3302_BonChua1_HMI" := 0.0; END_IF;
END_REGION

REGION Network 46: Sim Bồn Chứa 2: Giới hạn mức nước tối thiểu
   RUNG wire#powerrail
      Contact( "AI_HMI_Sim_Mode" )
      { S7_Templates := "SrcType := Real" } LT_Contact(in1 := "AI_LT3307_BonChua2_HMI", in2 := 0.0)
      { S7_GenerateENO := "TRUE" } Move(in := 0.0, out1 => "AI_LT3307_BonChua2_HMI")
   END_RUNG
   // the same network as SCL:
   IF "AI_HMI_Sim_Mode" AND ("AI_LT3307_BonChua2_HMI" < 0.0) THEN "AI_LT3307_BonChua2_HMI" := 0.0; END_IF;
END_REGION
END_ORGANIZATION_BLOCK
